         1630:	 //正极叠片升降移动至a等待高度 		  
	           			IF NOT DP_SinStepe THEN					
								 IF arrAxisCtrl[AxiseNo.AxisName.AnDTCarryingUpDown].Status.Homed AND arrAxisCtrl[AxiseNo.AxisName.AnDTCarryingUpDown].Status.NoMoving AND 
									NOT arrAxisCtrl[AxiseNo.AxisName.AnDTCarryingUpDown].Status.Error AND arrAxisCtrl[AxiseNo.AxisName.AnDTCarryingLine].Cmd.arrbRealPoint[2] AND
										 arrAxisCtrl[AxiseNo.AxisName.LeftYDUpDown].Cmd.arrbRealPoint[1] AND arrAxisCtrl[AxiseNo.AxisName.RightYDLine].Cmd.arrbRealPoint[2]     THEN
										IF arrAxisCtrl[AxiseNo.AxisName.AnDTCarryingUpDown].Cmd.arrbRealPoint[4] THEN
											arrAxisCtrl[AxiseNo.AxisName.AnDTCarryingUpDown].Cmd.iGoSetPos:=0;
										ELSE
											arrAxisCtrl[AxiseNo.AxisName.AnDTCarryingUpDown].Cmd.iGoSetPos:=4;//正极叠片升降移动至等待高度
										END_IF
								END_IF 
                                (*
								IF 	arrAxisCtrl[AxiseNo.AxisName.RightYDUpDown].Status.Homed AND arrAxisCtrl[AxiseNo.AxisName.RightYDUpDown].Status.NoMoving THEN
									IF arrAxisCtrl[AxiseNo.AxisName.RightYDUpDown].Cmd.arrbRealPoint[1] THEN
										arrAxisCtrl[AxiseNo.AxisName.RightYDUpDown].Cmd.iGoSetPos:=0;
									ELSE
										arrAxisCtrl[AxiseNo.AxisName.RightYDUpDown].Cmd.iGoSetPos:=1;//右压刀升降上升至初始高度
									END_IF
								END_IF													
  	                            *)
								IF arrAxisCtrl[AxiseNo.AxisName.AnDTCarryingUpDown].Cmd.arrbRealPoint[4] AND arrAxisCtrl[AxiseNo.AxisName.RightYDUpDown].Cmd.arrbRealPoint[15] AND
                                    arrAxisCtrl[AxiseNo.AxisName.AnDTCarryingUpDown].Status.NoMoving  AND arrAxisCtrl[AxiseNo.AxisName.RightYDUpDown].Status.NoMoving    THEN
						         	DT_SingeMode();//单步选择
									An_OverNGStep:=1670;
								END_IF		
                       END_IF	   						
 (*
  		1640://	压刀升降上升至初始高度	
					IF NOT DP_SinStepe THEN								
								IF 	arrAxisCtrl[AxiseNo.AxisName.RightYDUpDown].Status.Homed AND arrAxisCtrl[AxiseNo.AxisName.RightYDUpDown].Status.NoMoving THEN
									IF arrAxisCtrl[AxiseNo.AxisName.RightYDUpDown].Cmd.arrbRealPoint[1] THEN
										arrAxisCtrl[AxiseNo.AxisName.RightYDUpDown].Cmd.iGoSetPos:=0;
									ELSE
										arrAxisCtrl[AxiseNo.AxisName.RightYDUpDown].Cmd.iGoSetPos:=1;//右压刀升降上升至初始高度
									END_IF
								END_IF				
								IF arrAxisCtrl[AxiseNo.AxisName.RightYDUpDown].Cmd.arrbRealPoint[1] THEN
							     	DT_SingeMode();//单步选择
									An_OverNGStep:=1641;
								END_IF
						END_IF	   
	
		1641://	右压刀开合移至初始位		
			       IF NOT DP_SinStepe THEN
								IF 	arrAxisCtrl[AxiseNo.AxisName.RightYDLine].Status.Homed AND arrAxisCtrl[AxiseNo.AxisName.RightYDLine].Status.NoMoving THEN
										IF arrAxisCtrl[AxiseNo.AxisName.RightYDLine].Cmd.arrbRealPoint[1] THEN
											arrAxisCtrl[AxiseNo.AxisName.RightYDLine].Cmd.iGoSetPos:=0;
											DT_SingeMode();//单步选择
											An_OverNGStep:=1650;
										ELSE
											arrAxisCtrl[AxiseNo.AxisName.RightYDLine].Cmd.iGoSetPos:=1;//右压刀开合至初始位
										END_IF		
                                END_IF;	
					END_IF;				
					
		   	1650://右压刀升降下降至初始位，压隔膜			
					  IF NOT DP_SinStepe THEN
	                         	IF 	arrAxisCtrl[AxiseNo.AxisName.RightYDUpDown].Status.Homed AND arrAxisCtrl[AxiseNo.AxisName.RightYDUpDown].Status.NoMoving THEN
										IF arrAxisCtrl[AxiseNo.AxisName.RightYDUpDown].Cmd.arrbRealPoint[1] THEN
											arrAxisCtrl[AxiseNo.AxisName.RightYDUpDown].Cmd.iGoSetPos:=0;
									     	DT_SingeMode();//单步选择
									    	An_OverNGStep:=1670;
										ELSE
											arrAxisCtrl[AxiseNo.AxisName.RightYDUpDown].Cmd.iGoSetPos:=1;//右压刀升降轴下降至初始高度
										END_IF
									END_IF							  
					  
					  END_IF					   
					   
		     //1660:	 //判断真空					   
	*)

           1670://判断主轴是否停止、是否在初始位、是否有轴在耦合中
					IF NOT DP_SinStepe THEN
								IF arrAxis[AxiseNo.VirAxisName.VirMain].Status.NotMoving AND arrAxis[AxiseNo.VirAxisName.VirMain].NcToPlc.SetPos=0 AND NOT DT_AxiseCoupling THEN
									DT_SingeMode();//单步选择
									An_OverNGStep:=1691;
								ELSE
									DP_Step1:=100;//调用主轴回初始位子程序
									DT_SingeMode();//单步选择
									An_OverNGStep:=1690;
								END_IF
			    	END_IF		
			1690://判断主轴的模长的当前位置是否为0
				IF NOT DP_SinStepe THEN
					IF DP_Step1=6666 AND arrAxis[AxiseNo.VirAxisName.VirMain].Status.NotMoving AND arrAxis[AxiseNo.VirAxisName.VirMain].NcToPlc.SetPos=0 AND NOT DT_AxiseCoupling  THEN
						DT_SingeMode();//单步选择
						An_OverNGStep:=1691;
					END_IF	
				END_IF				
		1691:
			    IF 	arrAxisCtrl[AxiseNo.AxisName.LeftYDUpDown].Cmd.arrbRealPoint[1] AND (arrAxisCtrl[AxiseNo.AxisName.RightYDUpDown].Cmd.arrbRealPoint[1] OR arrAxisCtrl[AxiseNo.AxisName.RightYDUpDown].Cmd.arrbRealPoint[15] ) AND
					    arrCyCtrl[arrCyNo.CylinderName.AnScrapbinCy].Status.ONState  AND arrCyCtrl[arrCyNo.CylinderName.CaScrapbinUDCy].Status.OFFState AND
                        arrCyCtrl[arrCyNo.CylinderName.PoleHotCutterCy].Status.OFFState   THEN
					An_OverNGStep:=1695;
				END_IF	
		
		    1695://				
					IF An_CarryingPos2 THEN//正极在叠片位
							An_OverNGStep:=1700;//
					ELSIF An_CarryingPos1  THEN//正极在取片位
							 An_OverNGStep:=1800;//
					ELSE
						  DTPosError[11]:=TRUE;//踢正极对齐度NG片 时，正极取片即不在取片位，也不在叠片位
					END_IF;
		
	

	        1800://	调用正极NG踢废		
                    DT_TON[2].IN:=FALSE;	
					CCD.Over.Start.iPhotoDo:=2;
					CCD.Over.Finish.OverhandResult:=0;
					Mach_Control.DT_b.OverhandResult:=0;
					Mach_Control.DT_b.CDD_OverStart:=TRUE;
					
			        Mach_Control.An_b.An_Quantited:=Mach_Control.An_b.An_Quantited-1;//正极已叠片数减一
                    An_Step2:=10; 
                    An_OverNGStep:=1810;

			1810://判断负极叠台搬运是否有片，有片的话放到纠偏台
			         DT_TON[2].IN:=TRUE;	
						IF arrCyCtrl[arrCyNo.ElectValveName.CaDTCarryingVacuum].Io.DIOnSwitch AND  Mach_Control.Ca_b.Ca_DPCarryingFalg  THEN//负极再取片位且叠台搬运有片,把当前片放到纠偏台
							An_OverNGStep:=1820;
						ELSE
							An_OverNGStep:=1850;	
						END_IF
	
			1820://纠偏台回初始位
				//纠偏平台X1移动至初始位
				IF NOT DP_SinStepe THEN
					IF arrAxisCtrl[AxiseNo.AxisName.CadeviationX1].Status.Homed  AND arrAxisCtrl[AxiseNo.AxisName.CadeviationX1].Status.NoMoving AND NOT  arrAxisCtrl[AxiseNo.AxisName.CadeviationX1].Status.Error THEN
						IF arrAxisCtrl[AxiseNo.AxisName.CadeviationX1].Cmd.arrbRealPoint[1] THEN
							arrAxisCtrl[AxiseNo.AxisName.CadeviationX1].Cmd.iGoSetPos:=0;
						ELSE
							arrAxisCtrl[AxiseNo.AxisName.CadeviationX1].Cmd.iGoSetPos:=1;
						END_IF					
					END_IF
					//纠偏平台X2移动至初始位
					IF arrAxisCtrl[AxiseNo.AxisName.CadeviationX2].Status.Homed  AND arrAxisCtrl[AxiseNo.AxisName.CadeviationX2].Status.NoMoving AND NOT  arrAxisCtrl[AxiseNo.AxisName.CadeviationX2].Status.Error THEN
						IF arrAxisCtrl[AxiseNo.AxisName.CadeviationX2].Cmd.arrbRealPoint[1] THEN
							arrAxisCtrl[AxiseNo.AxisName.CadeviationX2].Cmd.iGoSetPos:=0;
						ELSE
							arrAxisCtrl[AxiseNo.AxisName.CadeviationX2].Cmd.iGoSetPos:=1;
						END_IF					
					END_IF
					//纠偏平台X2移动至初始位
					IF arrAxisCtrl[AxiseNo.AxisName.CadeviationY].Status.Homed  AND arrAxisCtrl[AxiseNo.AxisName.CadeviationY].Status.NoMoving AND NOT  arrAxisCtrl[AxiseNo.AxisName.CadeviationY].Status.Error THEN
						IF arrAxisCtrl[AxiseNo.AxisName.CadeviationY].Cmd.arrbRealPoint[1] THEN
							arrAxisCtrl[AxiseNo.AxisName.CadeviationY].Cmd.iGoSetPos:=0;
						ELSE
							arrAxisCtrl[AxiseNo.AxisName.CadeviationY].Cmd.iGoSetPos:=1;
						END_IF					
					END_IF
					IF arrAxisCtrl[AxiseNo.AxisName.CadeviationX1].Cmd.arrbRealPoint[1] AND arrAxisCtrl[AxiseNo.AxisName.CadeviationX2].Cmd.arrbRealPoint[1] AND arrAxisCtrl[AxiseNo.AxisName.CadeviationY].Cmd.arrbRealPoint[1] THEN
						DT_SingeMode();//单步选择	
						An_OverNGStep:=1830;	
						DT_TON[4].IN:=FALSE;
					END_IF	
				END_IF
			1830://叠台搬运极片放回纠偏台
				IF NOT DP_SinStepe THEN
					IF arrAxisCtrl[AxiseNo.AxisName.CaDTCarryingLine].Cmd.arrbRealPoint[1]  AND NOT Mach_Control.Ca_b.Ca_deviationFalg THEN 
						IF arrAxisCtrl[AxiseNo.AxisName.CaDTCarryingUpDown].Cmd.arrbRealPoint[2] THEN
							arrAxisCtrl[AxiseNo.AxisName.CaDTCarryingUpDown].Cmd.iGoSetPos:=0;
					    ELSE
							arrAxisCtrl[AxiseNo.AxisName.CaDTCarryingUpDown].Cmd.iGoSetPos:=2;//负极d叠台搬运下降至取片位
					    END_IF
                   END_IF
				       IF arrAxisCtrl[AxiseNo.AxisName.CaDTCarryingUpDown].Cmd.arrbRealPoint[2] THEN
				           	/// 吸盘破真空    纠偏台开真空
							arrCyCtrl[arrCyNo.ElectValveName.CaDTCarryingVacuum].Cmd.bON:=TRUE;	//负极叠台搬运升降真空	真空
							arrCyCtrl[arrCyNo.ElectValveName.CaDTCarryingVacuum].Cmd.bOFF:=FALSE;	//负极叠台搬运升降真空破真空								
							arrCyCtrl[arrCyNo.ElectValveName.CadeviationVacuum].Cmd.bON:=TRUE;	//负极纠偏台真空			
							arrCyCtrl[arrCyNo.ElectValveName.CadeviationVacuum].Cmd.bOFF:=FALSE;	//负极纠偏台真空	   
							DT_SingeMode();//单步选择	
							An_OverNGStep:=1840;
							DT_TON[4].IN:=TRUE;
							Mach_Control.Ca_b.Ca_deviationFalg:=TRUE;//置位位纠偏平台有料标记
							Mach_Control.Ca_b.Ca_DPCarryingFalg:=FALSE;//负极搬运真空吸盘有料标记复位
	                    END_IF
				END_IF
			1840://叠台搬运极片上升至凸轮耦合初始高度
				IF NOT DP_SinStepe THEN
					IF arrAxisCtrl[AxiseNo.AxisName.CaDTCarryingUpDown].Cmd.arrbRealPoint[4] AND DT_TON[4].Q THEN
						arrAxisCtrl[AxiseNo.AxisName.CaDTCarryingUpDown].Cmd.iGoSetPos:=0;
						/// 吸盘破真空    纠偏台开真空
						Mach_Control.Ca_b.Ca_deviationFalg:=TRUE;//置位位纠偏平台有料标记
						Mach_Control.Ca_b.Ca_DPCarryingFalg:=FALSE;//负极搬运真空吸盘有料标记复位
						Par.stDT_date.Ca_MQ_Slice[8]:=Par.stDT_date.Ca_MQ_Slice[9];
						DT_SingeMode();//单步选择	
						An_OverNGStep:=1850;
						DT_TON[4].IN:=FALSE;
					ELSE
						arrAxisCtrl[AxiseNo.AxisName.CaDTCarryingUpDown].Cmd.iGoSetPos:=4;//负极搬运升降2上升至凸轮耦合初始高度
					END_IF			
				END_IF		   
		

			
	        1860://等待正极NG踢废完成		
  
				
					 IF 	An_Step2=6666 THEN
						    An_OverNGStep:=0;
							DP_Step0:=0;
                           // An_OverNGMark:=FALSE;	
					 END_IF
	  END_CASE
END_IF

 CASE An_OverNGStep OF  
	 
		1850://
                  
				   IF Mach_Control.DT_b.OverhandResult<>3 AND  DT_TON[2].Q THEN
					  Mach_Control.An_b.Error[22]:=TRUE;//正极叠台搬运升降真空报警，电芯上有片，请拿掉 
				   END_IF
			
				 IF 	 Mach_Control.DT_b.OverhandResult=3 THEN
					     DT_TON[2].IN:=FALSE;	
						An_OverNGStep:=1860;
				 END_IF
 
 
 
 
     1200: //正到负取正极NG对其度片,	正极搬运与叠片各轴在初始位,负极在叠片位
	             VirMain_TON.IN:=FALSE;   
				//正到负_正极送片搬运平移轴凸轮耦合
				fbAnCamInCarryingLine.ParCamIn.SlaveScaling:=1;
				fbAnCamInCarryingLine.bCamInExecute:=TRUE;	
		    	fbAnCamInCarryingUpDown.iTableSel:=3;      //20240528SJ
                fbAnCamInCarryingUpDown.bCamInExecute:=TRUE;
			//正到负_正极叠片平移轴凸轮耦合
				fbAnCamInDTCarryingLine.ParCamIn.SlaveScaling:=1;
				fbAnCamInDTCarryingLine.bCamInExecute:=TRUE;			
                fbAnCamInDTCarryingUpDown.iTableSel:=3;   //  //20240528SJ
                fbAnCamInDTCarryingUpDown.bCamInExecute:=TRUE;
			//正到负_正极搬运旋转轴凸轮耦合		
				fbAnCamInCarryingWhirling.ParCamIn.SlaveScaling:=1;
				fbAnCamInCarryingWhirling.bCamInExecute:=TRUE;						
			
			//正到负_负极送片搬运平移轴凸轮耦合
				fbCaCamInCarryingLine2.ParCamIn.SlaveScaling:=-1;
				fbCaCamInCarryingLine2.bCamInExecute:=TRUE;
			   fbCaCamInCarryingUpDown2.iTableSel:=3; //20240528SJ
               fbCaCamInCarryingUpDown2.bCamInExecute:=TRUE;
			//正到负_负极叠片搬运平移轴凸轮耦合
				fbCaCamInDTCarryingLine.ParCamIn.SlaveScaling:=-1;
				fbCaCamInDTCarryingLine.bCamInExecute:=TRUE;
			    fbCaCamInDTCarryingUpDown.iTableSel:=3;  //20240528SJ
                fbCaCamInDTCarryingUpDown.bCamInExecute:=TRUE;
			//正到负_ 缓存轴轮耦合
				fbCamInGMBuffer2.iTableSel:=1;
				 fbCamInGMBuffer2.bCamInExecute:=TRUE;
			//正到负_隔膜平移轴凸轮耦合
				fbCamInGMDanserMove.iTableSel:=1;
				fbCamInGMDanserMove.bCamInExecute:=TRUE;
			
			//正到负_放卷虚轴凸轮耦合
				 fbCamInVirGMDriver2.iTableSel :=1;
				 fbCamInVirGMDriver2.bCamInExecute:=TRUE;		
					
					//判断凸轮是否耦合完成
						IF  fbAnCamInCarryingLine.bInSync  AND  fbAnCamInDTCarryingLine.bInSync AND fbAnCamInCarryingWhirling.bInSync AND 
							 fbCaCamInCarryingLine2.bInSync AND fbCaCamInDTCarryingLine.bInSync AND
							 fbCamInGMBuffer2.bInSync AND fbCamInGMDanserMove.bInSync AND 
							 fbCamInVirGMDriver2.bInSync   AND
							 fbAnCamInCarryingUpDown.bInSync AND fbAnCamInDTCarryingUpDown.bInSync AND fbCaCamInCarryingUpDown2.bInSync AND fbCaCamInDTCarryingUpDown.bInSync AND  
                            Mach_Control.U.DT_iMode=1  THEN
							An_OverNGStep:=1210;//
						ELSIF   fbAnCamInCarryingLine.bError  OR  fbAnCamInDTCarryingLine.bError OR 
							 fbCaCamInCarryingLine2.bError OR fbCaCamInDTCarryingLine.bError OR
							 fbCamInGMBuffer2.bError OR fbCamInGMDanserMove.bError OR 
							  fbAnCamInCarryingUpDown.bError OR fbAnCamInDTCarryingUpDown.bError OR fbCaCamInCarryingUpDown2.bError OR fbCaCamInDTCarryingUpDown.bError OR  
							 fbCamInVirGMDriver2.bError THEN
								Mach_Control.DT_b.Error[19]:=TRUE;//凸轮耦合报警
								An_OverNGStep:=9991;										
						END_IF		
			1210://主轴启动
									arrAxisCtrl[AxiseNo.VirAxisName.VirMain].Cmd	.bDynamitcsParSel:=2;
									arrAxisPar[AxiseNo.VirAxisName.VirMain].fTagatTime:=VirMain_TagatTime;
									arrAxisCtrl[AxiseNo.VirAxisName.VirMain].Cmd	.fPositon_of_Abs:=360;
									arrAxisCtrl[AxiseNo.VirAxisName.VirMain].Cmd	.bMoveAbs:=TRUE;		
									
									IF  arrAxis[AxiseNo.VirAxisName.VirMain].Status.Moving AND arrAxisCtrl[AxiseNo.VirAxisName.VirMain].Status.fActPos>=10  THEN
										VirMain_TON.IN:=FALSE;
										arrAxisCtrl[AxiseNo.VirAxisName.VirMain].Cmd	.bMoveAbs:=FALSE;	
										An_OverNGStep:=1500;	
									ELSE
										IF NOT VirMain_TON.Q THEN
											VirMain_TON.IN:=TRUE;
										ELSE
											VirMain_TON.IN:=FALSE;
											Mach_Control.DT_b.Error[22]:=TRUE;//主轴启动超时报警
											An_OverNGStep:=10001;	
									END_IF	
				 	    END_IF		

           1300: //正到负取正极NG对其度片,正极搬运与叠片各轴在初始位,, 负极在取片位,  隔膜平移在负极位
		              VirMain_TON.IN:=FALSE;
						//正到负_正极送片搬运平移轴凸轮耦合
					fbAnCamInCarryingLine.ParCamIn.SlaveScaling:=1;
					fbAnCamInCarryingLine.bCamInExecute:=TRUE;					
					fbAnCamInCarryingUpDown.iTableSel:=3;      //20240528SJ
					fbAnCamInCarryingUpDown.bCamInExecute:=TRUE;
				//正到负_正极叠片平移轴凸轮耦合
					fbAnCamInDTCarryingLine.ParCamIn.SlaveScaling:=1;
					fbAnCamInDTCarryingLine.bCamInExecute:=TRUE;		
					fbAnCamInDTCarryingUpDown.iTableSel:=3;   //  //20240528SJ
					fbAnCamInDTCarryingUpDown.bCamInExecute:=TRUE;

			//正到负_正极搬运旋转轴凸轮耦合		
				fbAnCamInCarryingWhirling.ParCamIn.SlaveScaling:=1;
				fbAnCamInCarryingWhirling.bCamInExecute:=TRUE;							
								
					//判断凸轮是否耦合完成
						IF  fbAnCamInCarryingLine.bInSync AND fbAnCamInDTCarryingLine.bInSync AND  fbAnCamInCarryingWhirling.bInSync  AND 
                            fbAnCamInCarryingUpDown.bInSync AND  fbAnCamInDTCarryingUpDown.bInSync AND 
                            Mach_Control.U.DT_iMode=1 THEN
							An_OverNGStep:=1310;//
						ELSIF fbAnCamInCarryingLine.bError OR  fbAnCamInDTCarryingLine.bError  OR   fbAnCamInCarryingUpDown.bError OR   fbAnCamInDTCarryingUpDown.bError   THEN
								Mach_Control.DT_b.Error[19]:=TRUE;//凸轮耦合报警
								An_OverNGStep:=9992;										
						END_IF			   
		   
			1310://主轴启动
									arrAxisCtrl[AxiseNo.VirAxisName.VirMain].Cmd	.bDynamitcsParSel:=2;
									arrAxisPar[AxiseNo.VirAxisName.VirMain].fTagatTime:=VirMain_TagatTime;
									arrAxisCtrl[AxiseNo.VirAxisName.VirMain].Cmd	.fPositon_of_Abs:=360;
									arrAxisCtrl[AxiseNo.VirAxisName.VirMain].Cmd	.bMoveAbs:=TRUE;			
						
									IF  arrAxis[AxiseNo.VirAxisName.VirMain].Status.Moving AND arrAxisCtrl[AxiseNo.VirAxisName.VirMain].Status.fActPos>=10  THEN
										VirMain_TON.IN:=FALSE;
										arrAxisCtrl[AxiseNo.VirAxisName.VirMain].Cmd	.bMoveAbs:=FALSE;	
										An_OverNGStep:=1500;	
									ELSE
										IF NOT VirMain_TON.Q THEN
											VirMain_TON.IN:=TRUE;
										ELSE
											VirMain_TON.IN:=FALSE;
											Mach_Control.DT_b.Error[22]:=TRUE;//主轴启动超时报警
											An_OverNGStep:=10002;	
									END_IF	
				 	    END_IF							
										
	       1400: //正到负取正极NG对其度片,正极搬运与叠片各轴在初始位,, 负极在取片位,  隔膜平移在正极位	
			              VirMain_TON.IN:=FALSE;
						//正到负_正极送片搬运平移轴凸轮耦合
						fbAnCamInCarryingLine.ParCamIn.SlaveScaling:=1;
						fbAnCamInCarryingLine.bCamInExecute:=TRUE;				
						fbAnCamInCarryingUpDown.iTableSel:=3;      //20240528SJ
						fbAnCamInCarryingUpDown.bCamInExecute:=TRUE;

					//正到负_正极叠片平移轴凸轮耦合
						fbAnCamInDTCarryingLine.ParCamIn.SlaveScaling:=1;
						fbAnCamInDTCarryingLine.bCamInExecute:=TRUE;
					   fbAnCamInDTCarryingUpDown.iTableSel:=3;   //  //20240528SJ
                       fbAnCamInDTCarryingUpDown.bCamInExecute:=TRUE;
						
						
					//正到负_正极搬运旋转轴凸轮耦合		
						fbAnCamInCarryingWhirling.ParCamIn.SlaveScaling:=1;
						fbAnCamInCarryingWhirling.bCamInExecute:=TRUE;						
						
					//正到负_ 缓存轴轮耦合
						fbCamInGMBuffer2.iTableSel:=1;
						 fbCamInGMBuffer2.bCamInExecute:=TRUE;
						 
					//正到负_隔膜平移轴凸轮耦合
						fbCamInGMDanserMove.iTableSel:=1;
						fbCamInGMDanserMove.bCamInExecute:=TRUE;
						
					//正到负_放卷虚轴凸轮耦合
						 fbCamInVirGMDriver2.iTableSel :=1;
						 fbCamInVirGMDriver2.bCamInExecute:=TRUE;			   
						
					//判断凸轮是否耦合完成
						IF   fbAnCamInCarryingLine.bInSync  AND  fbAnCamInDTCarryingLine.bInSync AND   fbAnCamInCarryingWhirling.bInSync AND
							 fbCamInGMBuffer2.bInSync AND fbCamInGMDanserMove.bInSync AND 
							 fbAnCamInCarryingUpDown.bInSync AND fbAnCamInDTCarryingUpDown.bInSync AND 
							 fbCamInVirGMDriver2.bInSync  AND 
                            Mach_Control.U.DT_iMode=1  THEN
							An_OverNGStep:=1410;//
						ELSIF  fbAnCamInCarryingLine.bError  OR  fbAnCamInDTCarryingLine.bError OR 
							     fbCamInGMBuffer2.bError OR fbCamInGMDanserMove.bError OR 
								 fbAnCamInCarryingUpDown.bError OR  fbAnCamInDTCarryingUpDown.bError OR
							     fbCamInVirGMDriver2.bError THEN
										Mach_Control.DT_b.Error[19]:=TRUE;//凸轮耦合报警
										An_OverNGStep:=9993;										
						END_IF		
	
			1410://主轴启动
									arrAxisCtrl[AxiseNo.VirAxisName.VirMain].Cmd	.bDynamitcsParSel:=2;
									arrAxisPar[AxiseNo.VirAxisName.VirMain].fTagatTime:=VirMain_TagatTime;
									arrAxisCtrl[AxiseNo.VirAxisName.VirMain].Cmd	.fPositon_of_Abs:=360;
									arrAxisCtrl[AxiseNo.VirAxisName.VirMain].Cmd	.bMoveAbs:=TRUE;					
									IF  arrAxis[AxiseNo.VirAxisName.VirMain].Status.Moving AND arrAxisCtrl[AxiseNo.VirAxisName.VirMain].Status.fActPos>=10  THEN
										VirMain_TON.IN:=FALSE;
										arrAxisCtrl[AxiseNo.VirAxisName.VirMain].Cmd	.bMoveAbs:=FALSE;	
										An_OverNGStep:=1500;	
									ELSE
										IF NOT VirMain_TON.Q THEN
											VirMain_TON.IN:=TRUE;
										ELSE
											VirMain_TON.IN:=FALSE;
											Mach_Control.DT_b.Error[22]:=TRUE;//主轴启动超时报警
											An_OverNGStep:=10003;	
									END_IF	
				 	    END_IF							
   
			1500://
				(*IF 	arrAxisCtrl[AxiseNo.VirAxisName.VirMain].Status.fActPos>230 AND  arrAxisCtrl[AxiseNo.VirAxisName.VirMain].Status.fActPos<240 AND Mach_Control.Ca_b.Ca_DPCarryingFalg  THEN//198
					IF Mach_Control.DT_b.DT_CCD_TwoModel THEN
							CCD.CaRec.Finish.RectifyX1:=0;
							CCD.CaRec.Finish.RectifyX2:=0;
							CCD.CaRec.Finish.RectifyY:=0;		
							CCD.CaRec.Finish.RectifyResult:=0;//拍照结果清零									
							Mach_Control.Ca_b.Ca_CCDStart :=TRUE;//启动CCD拍照
							CCD.CaRec.Start.iPhotoDo:=2;//启动CCD第二次拍照									
					END_IF			
				END_IF	*)		
				
				IF arrAxis[AxiseNo.VirAxisName.VirMain].NcToPlc.SetPos=360 AND  arrAxis[AxiseNo.VirAxisName.VirMain].Status.NotMoving  THEN
					DP_Step1:=100;//解除耦合，主轴回零子程序			
					An_OverNGStep:=1510;	
				END_IF	
			1510://			
				IF NOT DP_SinStepe THEN
					IF DP_Step1=6666 AND arrAxis[AxiseNo.VirAxisName.VirMain].Status.NotMoving AND arrAxis[AxiseNo.VirAxisName.VirMain].NcToPlc.SetPos=0 AND NOT DT_AxiseCoupling  THEN
						DT_SingeMode();//单步选择
						An_OverNGStep:=1600;
					END_IF	
				END_IF	

		    1700://	/踢正极NG对齐度片回正极取片位,(正极轴不动 ) ,正极搬运叠片各轴在叠片位		
			         VirMain_TON.IN:=FALSE;
					//负到正_正极搬运平移轴凸轮耦合
					fbAnCamInCarryingLine.ParCamIn.SlaveScaling:=-1;
					fbAnCamInCarryingLine.bCamInExecute:=TRUE;
					fbAnCamInCarryingUpDown.iTableSel:=3;      //20240528SJ
                   fbAnCamInCarryingUpDown.bCamInExecute:=TRUE;
					
					//负到正_正极叠片平移轴凸轮耦合
					fbAnCamInDTCarryingLine.ParCamIn.SlaveScaling:=-1;
					fbAnCamInDTCarryingLine.bCamInExecute:=TRUE;	
					fbAnCamInDTCarryingUpDown.iTableSel:=3;   //  //20240528SJ
					fbAnCamInDTCarryingUpDown.bCamInExecute:=TRUE;

					//负到正_正极搬运旋转轴凸轮耦合
						fbAnCamInCarryingWhirling.ParCamIn.SlaveScaling:=-1;
						fbAnCamInCarryingWhirling.bCamInExecute:=TRUE;								
				
				IF fbAnCamInCarryingLine.bInSync  AND 
					fbAnCamInDTCarryingLine.bInSync  AND
					fbAnCamInCarryingWhirling.bInSync AND  
                    fbAnCamInCarryingUpDown.bInSync AND   fbAnCamInDTCarryingUpDown.bInSync AND  
                    Mach_Control.U.DT_iMode=1  THEN   
					DT_SingeMode();//单步选择		
					An_OverNGStep:=1710;
				ELSIF fbAnCamInCarryingLine.bError OR //  fbCaCamInCarryingUpDown2.bError or
					  fbAnCamInDTCarryingLine.bError  OR  fbAnCamInCarryingUpDown.bError OR    fbAnCamInDTCarryingUpDown.bError   THEN   
					Mach_Control.DT_b.Error[19]:=TRUE;//凸轮耦合报警
					An_OverNGStep:=9994;
				END_IF		

				1710://主轴启动
				      				
									arrAxisCtrl[AxiseNo.VirAxisName.VirMain].Cmd	.bDynamitcsParSel:=2;
									arrAxisPar[AxiseNo.VirAxisName.VirMain].fTagatTime:=VirMain_TagatTime;
									arrAxisCtrl[AxiseNo.VirAxisName.VirMain].Cmd	.fPositon_of_Abs:=360;
									arrAxisCtrl[AxiseNo.VirAxisName.VirMain].Cmd	.bMoveAbs:=TRUE;			
						IF  arrAxis[AxiseNo.VirAxisName.VirMain].Status.Moving AND arrAxisCtrl[AxiseNo.VirAxisName.VirMain].Status.fActPos>=10  THEN
							VirMain_TON.IN:=FALSE;
							arrAxisCtrl[AxiseNo.VirAxisName.VirMain].Cmd	.bMoveAbs:=FALSE;	
							An_OverNGStep:=1720;	
						ELSE
								IF NOT VirMain_TON.Q THEN
									VirMain_TON.IN:=TRUE;
								ELSE
									VirMain_TON.IN:=FALSE;
									Mach_Control.DT_b.Error[22]:=TRUE;//主轴启动超时报警
									An_OverNGStep:=10004;	
							END_IF	
					   END_IF				

			1720://
				IF arrAxis[AxiseNo.VirAxisName.VirMain].NcToPlc.SetPos=360 AND  arrAxis[AxiseNo.VirAxisName.VirMain].Status.NotMoving  THEN
					DP_Step1:=100;//解除耦合，主轴回零子程序			
					An_OverNGStep:=1730;	
				END_IF	
	
				
			1730://			
				IF NOT DP_SinStepe THEN
					IF DP_Step1=6666 AND arrAxis[AxiseNo.VirAxisName.VirMain].Status.NotMoving AND arrAxis[AxiseNo.VirAxisName.VirMain].NcToPlc.SetPos=0 AND NOT DT_AxiseCoupling  THEN
						DT_SingeMode();//单步选择
						An_OverNGStep:=1800;
					END_IF	
				END_IF	
									
 END_CASE
END_ACTION

ACTION An_Rectifydev:
rAnCCD_Ton(IN:= , PT:=T#1.5S , Q=> , ET=> );//正极CCD拍照超时报警
IF (NOT Mach_Control.An_b.An_deviationFalg AND Mach_Control.U.DT_iMode=1) AND NOT Mach_Control.An_b.Demarcateing   THEN
//IF NOT Mach_Control.An_b.An_deviationFalg THEN
	Mach_Control.An_b.RectifydevDone:=FALSE;
	An_CCD_Done:=FALSE;
	CCD.AnRec.Finish.RectifyX1:=0;
	CCD.AnRec.Finish.RectifyX2:=0;
	CCD.AnRec.Finish.RectifyY:=0;
END_IF

rAnCCD_Ton1(IN:=Mach_Control.An_b.An_CCDStart , PT:=T#0.1S , Q=> , ET=> );//正极CCD拍照启动复位
IF rAnCCD_Ton1.Q THEN
	Mach_Control.An_b.An_CCDStart :=FALSE;
END_IF


An_CQ_ton(IN:=arrCyCtrl[arrCyNo.ElectValveName.AndeviationIonizedWind].Io.DOStatus1 , PT:=T#0.3S , Q=> , ET=>);
IF An_CQ_ton.Q THEN
	Mach_Control.An_b.An_Rectifydev_CQ:=FALSE;
	arrCyCtrl[arrCyNo.ElectValveName.AndeviationIonizedWind].Cmd.bON:=FALSE;//正极纠偏平台除尘
	arrCyCtrl[arrCyNo.ElectValveName.AndeviationIonizedWind].Cmd.bOFF:=TRUE;//正极纠偏平台除尘
END_IF



IF rAnUse[2].Q THEN
	CCD.AnRec.Finish.RectifyResult:=0;
	CCD.AnRec.Finish.RectifyX1:=0;
	CCD.AnRec.Finish.RectifyX2:=0;
	CCD.AnRec.Finish.RectifyY:=0;												
END_IF



IF Mach_Control.U.DT_iMode=1 THEN//在自动状态下
//判断负极是否允许取纠偏
IF (Mach_Control.An_b.An_deviationFalg AND (An_CCD_Done OR Mach_Control.An_b.RectifydevDone)) (*AND CCD.AnRec.Finish.RectifyResult=1 AND Mach_Control.An_b.RectifydevDone)*) OR
	 (Mach_Control.An_b.An_deviationFalg AND CCD.AnRec.Finish.RectifyResult<>1 AND arrAxisCtrl[AxiseNo.AxisName.AndeviationX1].Cmd.arrbRealPoint[1] AND 	arrAxisCtrl[AxiseNo.AxisName.AndeviationX2].Cmd.arrbRealPoint[1]  AND 	arrAxisCtrl[AxiseNo.AxisName.AndeviationY].Cmd.arrbRealPoint[1] )OR
	(Mach_Control.U.CCD_ChosesHMI  OR Mach_Control.U.EmptyRunMode)	 THEN
	Mach_Control.An_b.An_deviationDPOK:=TRUE;//取正极 偏平台极片允许
ELSE
	Mach_Control.An_b.An_deviationDPOK:=FALSE;
END_IF 	

	CASE An_StandbyStep0 OF
			0://判断正极纠偏平台是否有极片
				IF Mach_Control.An_b.An_deviationFalg AND NOT Mach_Control.U.EmptyRunMode  THEN
						IF NOT An_CCD_Done THEN
							CCD.AnRec.Finish.RectifyResult:=0;
							CCD.AnRec.Finish.RectifyX1:=0;
							CCD.AnRec.Finish.RectifyX2:=0;
							CCD.AnRec.Finish.RectifyY:=0;
							iMD11:=1;
							An_StandbyStep0:=10;
						END_IF
				ELSE
						iMD11:=2;
						An_RecdevPla_Step0:=0;
						Mach_Control.An_b.RectifydevStart :=FALSE;
						An_StandbyStep0:=10;
				END_IF
			10://正极纠偏平台回初始位
			IF  NOT Mach_Control.U.EmptyRunMode THEN
					Mach_Control.An_b.RectifydevStart :=FALSE;//复位纠偏启动
					Mach_Control.An_b.RectifydevDone:=FALSE;//复位纠偏完成
					IF Mach_Control.An_b.CarryingSafepos[4] THEN
							//纠偏平台X1移动至初始位
							IF arrAxisCtrl[AxiseNo.AxisName.AndeviationX1].Status.Homed  AND arrAxisCtrl[AxiseNo.AxisName.AndeviationX1].Status.NoMoving AND NOT  arrAxisCtrl[AxiseNo.AxisName.AndeviationX1].Status.Error THEN
								IF arrAxisCtrl[AxiseNo.AxisName.AndeviationX1].Cmd.arrbRealPoint[1] THEN
									arrAxisCtrl[AxiseNo.AxisName.AndeviationX1].Cmd.iGoSetPos:=0;
								ELSE
									arrAxisCtrl[AxiseNo.AxisName.AndeviationX1].Cmd.iGoSetPos:=1;
								END_IF					
							END_IF
							//纠偏平台X2移动至初始位
							IF arrAxisCtrl[AxiseNo.AxisName.AndeviationX2].Status.Homed  AND arrAxisCtrl[AxiseNo.AxisName.AndeviationX2].Status.NoMoving AND NOT  arrAxisCtrl[AxiseNo.AxisName.AndeviationX2].Status.Error THEN
								IF arrAxisCtrl[AxiseNo.AxisName.AndeviationX2].Cmd.arrbRealPoint[1] THEN
									arrAxisCtrl[AxiseNo.AxisName.AndeviationX2].Cmd.iGoSetPos:=0;
								ELSE
									arrAxisCtrl[AxiseNo.AxisName.AndeviationX2].Cmd.iGoSetPos:=1;
								END_IF					
							END_IF
							//纠偏平台X2移动至初始位
							IF arrAxisCtrl[AxiseNo.AxisName.AndeviationY].Status.Homed  AND arrAxisCtrl[AxiseNo.AxisName.AndeviationY].Status.NoMoving AND NOT  arrAxisCtrl[AxiseNo.AxisName.AndeviationY].Status.Error THEN
								IF arrAxisCtrl[AxiseNo.AxisName.AndeviationY].Cmd.arrbRealPoint[1] THEN
									arrAxisCtrl[AxiseNo.AxisName.AndeviationY].Cmd.iGoSetPos:=0;
								ELSE
									arrAxisCtrl[AxiseNo.AxisName.AndeviationY].Cmd.iGoSetPos:=1;
								END_IF					
							END_IF	
							IF 	 arrAxisCtrl[AxiseNo.AxisName.AndeviationX1].Cmd.arrbRealPoint[1] AND 	arrAxisCtrl[AxiseNo.AxisName.AndeviationX2].Cmd.arrbRealPoint[1]  AND 	arrAxisCtrl[AxiseNo.AxisName.AndeviationY].Cmd.arrbRealPoint[1] THEN
									IF  iMD11=1 THEN
											 An_StandbyStep0:=101;
											 rAnCCD_Ton.IN:=FALSE;
									 ELSIF  iMD11=2 THEN
											An_StandbyStep0:=0;
									 END_IF  			
							END_IF						
					END_IF
	END_IF
			101:
					CCD.AnRec.Finish.RectifyResult:=0;
					Mach_Control.An_b.An_CCDStart :=TRUE;//启动CCD拍照						
					CCD.AnRec.Start.iPhotoDo:=1;//第一次拍照	
					CCD.AnRec.Start.stPoleNo:=Par.stDT_date.An_MQ_Slice[1].stPoleNo;	
					An_StandbyStep0:=110;	
			110:
					IF NOT rAnCCD_Ton.Q THEN						
						rAnCCD_Ton.IN:=TRUE;
						IF Mach_Control.An_b.An_deviationCCDDone OR Mach_Control.U.CCD_ChosesHMI THEN
							rAnCCD_Ton.IN:=FALSE;
							An_CCD_Done:=TRUE;
							An_StandbyStep0:=111;
						END_IF
					ELSE
							rAnCCD_Ton.IN:=FALSE;
							Mach_Control.An_b.Error[7]:=TRUE;//正极CCD第一次拍照超时
							An_StandbyStep0:=9999;
					END_IF
			
			111://启动拍照			
					Mach_Control.An_b.An_CCDStart :=FALSE;//启动CCD拍照						
					rAnCCD_Ton.IN:=FALSE;
					An_StandbyStep0:=0;					

	END_CASE
ELSE
//正极纠偏平台CCD标定自动
IF Mach_Control.An_b.DemarcateStart THEN
	CCD.AnRec.Start.iPhotoDo:=1;//第一次拍照	
END_IF
An_Demarcate(
	Step0:=An_Demarcate_Step0,
	AxisX1_NO:=AxiseNo.AxisName.AndeviationX1 , //正极纠偏X1轴号
	AxisX2_NO:=AxiseNo.AxisName.AndeviationX2 , //正极纠偏X2轴号
	AxisY_NO:=AxiseNo.AxisName.AndeviationY , //正极纠偏Y轴号
	DemarcateStart:=Mach_Control.An_b.DemarcateStart , //纠偏平台CCD标定启动
	CCDStart:=Mach_Control.An_b.An_CCDStart , //CCD拍照启动
	CCDNo:=CCD.AnRec.iDemCount,//CCD拍照次数
	DemarcateResult:=CCD.AnRec.iDemarcatResult,//标定结果
	DemarcateDone:=Mach_Control.An_b.DemarcateDone ,//CCD标定完成
	Demarcateing:=Mach_Control.An_b.Demarcateing,	//CCD标定中
	Error :=Mach_Control.An_b.Error[8]  );//CCD标定NG
END_IF
//正极纠偏自动
rAn_RecdevPlaR_TRIG(CLK:=Mach_Control.An_b.An_deviationFalg AND (CCD.AnRec.Finish.RectifyResult=1 OR CCD.AnRec.Finish.RectifyResult=2 ) AND NOT Mach_Control.U.CCD_ChosesHMI AND NOT Mach_Control.An_b.RectifydevDone AND 
										 		(CCD.AnRec.Finish.RectifyX1<>0 OR CCD.AnRec.Finish.RectifyX2<>0 OR CCD.AnRec.Finish.RectifyY<>0) AND CCD.AnRec.Start.iPhotoDo=1  , Q=> );//AND NOT Mach_Control.An_b.An_VacuumErrorNG
IF rAn_RecdevPlaR_TRIG.Q  THEN//AND NOT Blueflaging
	Mach_Control.An_b.RectifydevStart:=TRUE;
END_IF

//纠偏结果限定
IF (CCD.AnRec.Finish.RectifyX1>=15 OR CCD.AnRec.Finish.RectifyX2>=15 OR CCD.AnRec.Finish.RectifyY>=10 OR
	CCD.AnRec.Finish.RectifyX1<=-15 OR CCD.AnRec.Finish.RectifyX2<=-15 OR CCD.AnRec.Finish.RectifyY<=-10) AND NOT Mach_Control.An_b.Demarcateing THEN
	CCD.AnRec.Finish.RectifyX1:=0;
	CCD.AnRec.Finish.RectifyX2:=0;
	CCD.AnRec.Finish.RectifyY:=0;
END_IF


CCD.AnRec.Finish.Offset_X:=fCaOffsetMean_X;
CCD.AnRec.Finish.Offset_Y:=fCaOffsetMean_Y;

An_RecdevPla(
	Step0:=An_RecdevPla_Step0,
	RecdevStart:=Mach_Control.An_b.RectifydevStart , //正极纠偏平台纠偏启动
	RecdevDone:=Mach_Control.An_b.RectifydevDone , //正极纠偏平台纠偏完成
	RecdevAgree:=Mach_Control.An_b.CarryingSafepos[4] , //正极纠偏平台纠偏允许
	AxisX1_NO:=AxiseNo.AxisName.AndeviationX1  , //正极纠偏平台X1轴号
	AxisX2_NO:=AxiseNo.AxisName.AndeviationX2 , //正极纠偏平台X2轴号
	AxisY_NO:=AxiseNo.AxisName.AndeviationY  , //正极纠偏平台Y轴号
	CCD_X1:=CCD.AnRec.Finish.RectifyX1 ,//正极纠偏平台X1纠偏量
	CCD_X2:=CCD.AnRec.Finish.RectifyX2 , //正极纠偏平台X2纠偏量
	CCD_Y:=CCD.AnRec.Finish.RectifyY );//正极纠偏平台Y纠偏量
	
//纠偏平台重复精度测试
AN_RectifyTry_fb(
	Execute:=Mach_Control.An_b.RectifyTryStart AND Mach_Control.U.DT_iMode=3 , //纠偏平台重复精度测试启动 
	AxisNO_X:=AxiseNo.AxisName.AndeviationX1 , 
	AxisNO_Y:= AxiseNo.AxisName.AndeviationX2, 
	AxisNO_R:=AxiseNo.AxisName.AndeviationY , 
	Demarcate_X:=Par.stDT_date.An_Demarcate_X , //纠偏平台重复精度测试X纠偏量
	Demarcate_Y:=Par.stDT_date.An_Demarcate_Y , //纠偏平台重复精度测试Y纠偏量
	Demarcate_R:=Par.stDT_date.An_Demarcate_R ,  //纠偏平台重复精度测试R纠偏量
	CCDNo:=Par.stDT_date.An_CCDNo, //纠偏平台重复精度测试次数
	CCDStart:= Mach_Control.An_b.An_CCDStart );
	
//吸盘重复精度测试		
An_SuckerTest_fb(
	Execute:=Mach_Control.An_b.SuckerTestStart AND Mach_Control.U.DT_iMode=3 , //吸盘重复精度测试启动 , 
	AxisNO_1:= AxiseNo.AxisName.AnDTCarryingUpDown, 
	AxisNO_2:=AxiseNo.AxisName.AnDTCarryingLine , 
	AxisNO_X:= AxiseNo.AxisName.AndeviationX1 , 
	AxisNO_Y:= AxiseNo.AxisName.AndeviationX2, 
	AxisNO_R:= AxiseNo.AxisName.AndeviationY , 
	DTCarryingVacuum:=arrCyNo.ElectValveName.AnDTCarryingVacuum , 
	deviationVacuum:= arrCyNo.ElectValveName.AndeviationVacuum, 
	deviationVacuumBark:=arrCyNo.ElectValveName.AndeviationVacuumBark, 
	CCDCount:= Par.stDT_date.An_CCDCount, //吸盘重复精度测试次数
	CCDStart:=Mach_Control.An_b.An_CCDStart,	
	CCD_X1:=CCD.AnRec.Finish.RectifyX1 ,//正极纠偏平台X1纠偏量
	CCD_X2:=CCD.AnRec.Finish.RectifyX2 , //正极纠偏平台X2纠偏量
	CCD_Y:=CCD.AnRec.Finish.RectifyY,//正极纠偏平台Y纠偏量
    DTiMode:= Mach_Control.U.DT_iMode  );
	
	//正极通讯监控
rtAn_CCDTest1(CLK:=Mach_Control.An_b.bAnCCD_TestDo , Q=> );
IF rtAn_CCDTest1.Q THEN
	bAn_CCDTest1:=FALSE;
	bAn_CCDTest2:=FALSE;
END_IF
IF Mach_Control.An_b.bAnCCD_TestDo THEN
	rtAn_CCDTest2(CLK:=Mach_Control.An_b.An_CCDStart , Q=> );
	rtAn_CCDTest3(CLK:=CCD.AnRec.Finish.RectifyResult<>0 , Q=> );
	rtAn_CCDTest4(CLK:=Mach_Control.An_b.An_deviationCCDDone , Q=> );
	IF rtAn_CCDTest2.Q THEN
		bAn_CCDTest1:=TRUE;
		bAn_CCDTest2:=TRUE;
		CCD.AnRec.Finish.RectifyResult:=0;
	END_IF
	IF rtAn_CCDTest3.Q THEN
		bAn_CCDTest1:=FALSE;
	END_IF	
	IF rtAn_CCDTest4.Q THEN
		bAn_CCDTest2:=FALSE;
	END_IF
	tonAn_CCDTest1(IN:=bAn_CCDTest1 , PT:=T#999MS , Q=> , ET=> );
	tonAn_CCDTest2(IN:=bAn_CCDTest2 , PT:=T#999MS , Q=> , ET=> );
	IF bAn_CCDTest1 THEN
		Mach_Control.An_b.iAnCCD_RectifyCT:= TIME_TO_INT(tonAn_CCDTest1.ET);
	END_IF
	IF bAn_CCDTest2 THEN
		Mach_Control.An_b.iAnCCD_PhotoCT:= TIME_TO_INT(tonAn_CCDTest2.ET);
	END_IF
	IF tonAn_CCDTest1.Q THEN
		Mach_Control.An_b.bAnCCD_TestDo:=FALSE;
	END_IF
END_IF
	
//正极白班NG计数
IF HMI_Hour>=8 AND HMI_Hour<20 AND An_Step2>50 AND An_Step2<70 THEN
  IF CCD.AnRec.Finish.NG_Code = 1 THEN
   CCD.AnRec.DayNgclassification.X1_NG :=CCD.AnRec.DayNgclassification.X1_NG+1 ;
   CCD.AnRec.Finish.NG_Code := 0 ;
  ELSIF CCD.AnRec.Finish.NG_Code = 2 THEN
   CCD.AnRec.DayNgclassification.X2_NG := CCD.AnRec.DayNgclassification.X2_NG+1 ;  
   CCD.AnRec.Finish.NG_Code := 0 ;
  ELSIF CCD.AnRec.Finish.NG_Code = 3 THEN
   CCD.AnRec.DayNgclassification.Y_NG := CCD.AnRec.DayNgclassification.Y_NG+1 ;  
   CCD.AnRec.Finish.NG_Code := 0 ;
  ELSIF CCD.AnRec.Finish.NG_Code = 4 THEN
   CCD.AnRec.DayNgclassification.R_NG := CCD.AnRec.DayNgclassification.R_NG+1 ;   
   CCD.AnRec.Finish.NG_Code := 0 ; 
  ELSIF CCD.AnRec.Finish.NG_Code = 5 THEN 
   CCD.AnRec.DayNgclassification.other_NG :=  CCD.AnRec.DayNgclassification.other_NG+1;
   CCD.AnRec.Finish.NG_Code := 0 ;
  END_IF	
END_IF  

DayClear1(CLK:=(HMI_Hour=8 AND HMI_Minute=0 AND HMI_Second=0 ) , Q=> );
NightClear1(CLK:=(HMI_Hour=20 AND HMI_Minute=0 AND HMI_Second=0) , Q=> );

//正极白班N清零
IF DayClear1.Q  THEN
  Par.stDT_date.An_Rectifydev_DayNG:=0;
END_IF 

IF CCD.AnRec.DayNgclassification.NgClear[1] OR DayClear1.Q  THEN
   CCD.AnRec.DayNgclassification.X1_NG :=0 ;
END_IF

IF CCD.AnRec.DayNgclassification.NgClear[2] OR DayClear1.Q  THEN
   CCD.AnRec.DayNgclassification.X2_NG :=0 ;
END_IF

IF CCD.AnRec.DayNgclassification.NgClear[3] OR DayClear1.Q  THEN
   CCD.AnRec.DayNgclassification.Y_NG :=0 ;
END_IF

IF CCD.AnRec.DayNgclassification.NgClear[4] OR DayClear1.Q  THEN
   CCD.AnRec.DayNgclassification.R_NG :=0 ;
END_IF	

IF CCD.AnRec.DayNgclassification.NgClear[5] OR DayClear1.Q  THEN
   CCD.AnRec.DayNgclassification.other_NG :=0 ;
END_IF	
	
//正极晚班NG计数
IF ((HMI_Hour>=0 AND HMI_Hour<8) OR  (HMI_Hour>=20 AND HMI_Hour<=23)) AND An_Step2>50 AND An_Step2<70  THEN
  IF CCD.AnRec.Finish.NG_Code = 1 THEN
   CCD.AnRec.NightNgclassification.X1_NG :=CCD.AnRec.NightNgclassification.X1_NG+1 ;
   CCD.AnRec.Finish.NG_Code := 0 ;
  ELSIF CCD.AnRec.Finish.NG_Code = 2 THEN
   CCD.AnRec.NightNgclassification.X2_NG := CCD.AnRec.NightNgclassification.X2_NG+1 ;  
   CCD.AnRec.Finish.NG_Code := 0 ;
  ELSIF CCD.AnRec.Finish.NG_Code = 3 THEN
   CCD.AnRec.NightNgclassification.Y_NG := CCD.AnRec.NightNgclassification.Y_NG+1 ;  
   CCD.AnRec.Finish.NG_Code := 0 ;
  ELSIF CCD.AnRec.Finish.NG_Code = 4 THEN
   CCD.AnRec.NightNgclassification.R_NG := CCD.AnRec.NightNgclassification.R_NG+1 ;   
   CCD.AnRec.Finish.NG_Code := 0 ; 
  ELSIF CCD.AnRec.Finish.NG_Code = 5 THEN 
   CCD.AnRec.NightNgclassification.other_NG :=  CCD.AnRec.NightNgclassification.other_NG+1;
   CCD.AnRec.Finish.NG_Code := 0 ;
  END_IF	
END_IF  

//正极晚班NG清零
IF  NightClear1.Q  THEN
   Par.stDT_date.An_Rectifydev_NightNG:=0;
END_IF

IF CCD.AnRec.NightNgclassification.NgClear[1] OR NightClear1.Q  THEN
   CCD.AnRec.NightNgclassification.X1_NG :=0 ;
END_IF

IF CCD.AnRec.NightNgclassification.NgClear[2] OR NightClear1.Q  THEN
   CCD.AnRec.NightNgclassification.X2_NG :=0 ;
END_IF

IF CCD.AnRec.NightNgclassification.NgClear[3] OR NightClear1.Q  THEN
   CCD.AnRec.NightNgclassification.Y_NG :=0 ;
END_IF

IF CCD.AnRec.NightNgclassification.NgClear[4] OR NightClear1.Q  THEN
   CCD.AnRec.NightNgclassification.R_NG :=0 ;
END_IF	

IF CCD.AnRec.NightNgclassification.NgClear[5] OR NightClear1.Q  THEN
   CCD.AnRec.NightNgclassification.other_NG :=0 ;
END_IF
END_ACTION

ACTION An_StandbyMain:
An_TON[1](PT:=T#0.5S);//正极拍照结果超时报警
An_TON[2](PT:=T#5S);//叠台主轴启动超时报警延时
An_TON[3](PT:=T#0.5S);
An_TON[5](PT:=T#10MS);
An_TON[6](PT:=T#0.2S);
An_TON[7](PT:=T#0.3S);
An_TON[8](PT:=T#0.3S);
An_TON[9](PT:=T#0.1S);
An_TON[10](PT:=T#2.5S);
An_TON[11](PT:=T#2.5S);
//An_StandbyStep1



IF Mach_Control.U.DT_iMode=1 THEN//在自动状态下	
	(**********************************************************************正极备料自动**********************************************************************************)
	CASE An_StandbyStep1 OF
	1000://处理负极片取 AND AN_CarryingPos1
		IF NOT DP_SinStepe THEN
			An_TON[7].IN:=TRUE;
			IF Mach_Control.An_b.An_CarryingFalg AND  Mach_Control.An_b.An_DPCarryingFalg AND  NOT Mach_Control.An_b.An_deviationFalg   AND 
			   ( CCD.AnRec.Finish.RectifyResult=1 OR Mach_Control.U.CCD_ChosesHMI	  OR Mach_Control.U.EmptyRunMode (*OR Blueflaging*)	)THEN	
					An_StandbyStep1:=6666;	//正极取料完成
			//正极搬运、叠台搬运、纠偏平台都无料---状态1
			ELSIF NOT Mach_Control.An_b.An_CarryingFalg AND  NOT Mach_Control.An_b.An_DPCarryingFalg AND NOT Mach_Control.An_b.An_deviationFalg  THEN   // 状态1  0   0    0		 	OK   				      	                             
				IF AN_CarryingPos1 THEN 
					An_StandbyStep1:=2000;//取流水线的极片	
				ELSIF AN_CarryingPos2 THEN 
					iND1:=3;
					An_StandbyStep1:=6000;//
				ELSIF (An_Step0=6666 OR An_Step0=0) AND ( An_Step3=6666 OR An_Step3=0) AND An_TON[7].Q THEN
					//Mach_Control.DT_b.Error[8]:=TRUE;//取正极片凸轮耦合时，正极取片轴不在取片位也不在叠片位报警
					An_StandbyStep1:=9993;
					AnPosError[1]:=TRUE;
				END_IF		
			//正极搬运吸盘有料，叠台搬运、纠偏台无料----状态2
			ELSIF Mach_Control.An_b.An_CarryingFalg AND  NOT Mach_Control.An_b.An_DPCarryingFalg AND  NOT Mach_Control.An_b.An_deviationFalg AND   Mach_Control.Ca_b.Ca_Quantited<>0 THEN  // 状态2  1  0  0		
				IF AN_CarryingPos1 THEN  		
					IF Mach_Control.An_b.An_deviationFPOK   THEN//需要判断热切横移轴在安全位
						DT_SingeMode();//单步选择		
						iND1:=1;	
						An_StandbyStep1:=6000;//通过凸轮耦合放极片到纠偏平台
					END_IF
				ELSIF AN_CarryingPos2  THEN			
					An_StandbyStep1:=2500;//  负极送片搬运放片到纠偏台					      					
				ELSIF (An_Step0=6666 OR An_Step0=0)  AND ( An_Step3=6666 OR An_Step3=0) AND An_TON[7].Q THEN
					//Mach_Control.DT_b.Error[8]:=TRUE;//叠负极片凸轮耦合时，负极取片轴不在耦合位报警
					An_StandbyStep1:=9993;
					AnPosError[2]:=TRUE;									   										 
				END_IF	
			//正极搬运、叠台搬运无料，纠偏台有料----状态3	
			ELSIF NOT Mach_Control.An_b.An_CarryingFalg AND  NOT Mach_Control.An_b.An_DPCarryingFalg AND  Mach_Control.An_b.An_deviationFalg THEN // 状态3    0  0  1
				IF AN_CarryingPos1 THEN  									
					IF (CCD.AnRec.Finish.RectifyResult=1 OR  Mach_Control.U.CCD_ChosesHMI OR Mach_Control.U.EmptyRunMode  (*OR  Blueflaging *))  THEN								        	
						An_TON[1].IN:=FALSE;				
						An_StandbyStep1:=2100;//取流水线的极片、同时取纠偏平台的极片
					ELSIF CCD.AnRec.Finish.RectifyResult=2 OR CCD.AnRec.Finish.RectifyResult= 3 OR CCD.AnRec.Finish.RectifyResult= 4  THEN
						//   DT_SingeMode();//单步选择			
						An_TON[1].IN:=FALSE;			
						An_StandbyStep1:=2200;//取纠偏平台的极片，再踢纠偏平台的NG片，同时取流水线的片
					ELSE
						IF NOT An_TON[1].Q THEN
							An_TON[1].IN:=TRUE;
						ELSE
							An_TON[1].IN:=FALSE;
							Mach_Control.An_b.Error[36]:=TRUE;//正极CCD第一次拍照超时
							An_StandbyStep1:=9999;
						END_IF
					END_IF
				ELSIF  AN_CarryingPos2 THEN
					IF Mach_Control.An_b.An_deviationDPOK   THEN//   
						DT_SingeMode();//单步选择		
						iND1:=2;	
						An_StandbyStep1:=6000;//通过凸轮耦合放极片到纠偏平台
					END_IF
				ELSIF (An_Step0=6666 OR An_Step0=0)  AND ( An_Step3=6666 OR An_Step3=0) AND An_TON[7].Q THEN
					//Mach_Control.DT_b.Error[8]:=TRUE;//叠负极片凸轮耦合时，负极取片轴不在耦合位报警
					 An_StandbyStep1:=9993;
					 AnPosError[3]:=TRUE;
				END_IF		
			//正极搬运吸盘有料，叠台搬运无料，纠偏台有料-----状态4
			ELSIF Mach_Control.An_b.An_CarryingFalg AND  NOT Mach_Control.An_b.An_DPCarryingFalg AND   Mach_Control.An_b.An_deviationFalg  THEN 
				IF Mach_Control.An_b.An_deviationDPOK AND arrAxisCtrl[AxiseNo.AxisName.AnDTCarryingLine].Cmd.arrbRealPoint[1]AND 
					arrAxisCtrl[AxiseNo.AxisName.AnDTCarryingLine].Status.Homed AND arrAxisCtrl[AxiseNo.AxisName.AnDTCarryingLine].Status.NoMoving
					AND (An_Step3=6666 OR An_Step3=0) THEN				
					An_StandbyStep1:=4000;//单独取纠偏平台
					An_Step3:=10;	
				END_IF
			//正极搬运吸盘无料，叠台搬运有纠偏OK料，纠偏平台无料-----状态5，流水取料且不丢NG
			ELSIF  ( Mach_Control.An_b.An_DPCarryingFalg AND  CCD.AnRec.Finish.RectifyResult=1 OR Mach_Control.U.EmptyRunMode OR  Mach_Control.U.CCD_ChosesHMI(* OR  Blueflaging*)	) AND NOT  Mach_Control.An_b.An_deviationFalg AND (An_Step0=6666 OR An_Step0=0) THEN// 状态4 正常       0 (1)     1 0    				
				IF  AN_CarryingPos1 THEN   
					IF  NOT Mach_Control.An_b.An_CarryingFalg THEN
						An_StandbyStep1:=2000;//取流水线的极片		
					END_IF
				ELSIF    An_TON[7].Q THEN// ------------------------20231209新增(An_Step0=6666 OR An_Step0=0)  AND
					  //Mach_Control.DT_b.Error[8]:=TRUE;//叠负极片凸轮耦合时，负极取片轴不在耦合位报警
					   An_StandbyStep1:=9993;
					   AnPosError[4]:=TRUE;
				END_IF			
			//	正极搬运吸盘无料，叠台搬运有纠偏NG料，纠偏台无料----状态6，取流水线极片且叠台搬运丢NG片			
			ELSIF  ( Mach_Control.An_b.An_DPCarryingFalg AND  CCD.AnRec.Finish.RectifyResult<>1 ) AND  NOT  Mach_Control.An_b.An_deviationFalg AND  NOT    Mach_Control.U.CCD_ChosesHMI AND (An_Step0=6666 OR An_Step0=0) THEN			// 状态5        0 (1)     1 0    
				   IF  AN_CarryingPos1 THEN      		
					  IF  NOT Mach_Control.an_b.An_CarryingFalg THEN    
						An_StandbyStep1:=2300;//踢纠偏平台的NG片，同时取流水线的片	     
					  ELSIF   Mach_Control.an_b.An_CarryingFalg THEN     
						An_StandbyStep1:=2400;//踢纠偏平台的NG片，同时取流水线的片	    
					  END_IF      
				   ELSIF   An_TON[7].Q THEN// ------------------------20231209新增(An_Step0=6666 OR An_Step0=0)
					  //Mach_Control.DT_b.Error[8]:=TRUE;//叠负极片凸轮耦合时，负极取片轴不在耦合位报警
					   An_StandbyStep1:=9993;
					   AnPosError[5]:=TRUE;
				  END_IF				
			END_IF	
		END_IF
	//取料流程调用				
	2000://调用取流水线子程序
		IF NOT DP_SinStepe THEN
			IF An_Step0=0 OR An_Step0=6666 THEN
				An_Step0:=10;//正极取流水线子程序
			END_IF
			DT_SingeMode();//单步选择		
			An_StandbyStep1:=2010;	
		END_IF	
	2010://判断取料是否完成
		IF An_Step0=6666 THEN
			DT_SingeMode();//单步选择		
			An_StandbyStep1:=1000;	
		END_IF				
	2100://调用取流水线子程序，取纠偏极片子程序
		IF NOT DP_SinStepe THEN
			IF An_Step0=0 OR An_Step0=6666 THEN
				An_Step0:=10;//正极取流水线子程序
			END_IF
				An_Step3:=10;//正极取纠偏平台子程序
				DT_SingeMode();//单步选择					
				An_StandbyStep1:=2110;	
		END_IF
	2110://判断正极取片流水线的极片、取纠偏平台的极片是否完成
		IF NOT DP_SinStepe THEN
			IF 	An_Step0=6666 AND 	An_Step3=6666 THEN
				DT_SingeMode();//单步选择							
				An_StandbyStep1:=1000;	
			END_IF
		END_IF			
	2200://先取纠偏平台的极片，同时根据条件判断是否可以取流水线的极片
		IF NOT DP_SinStepe THEN
			An_Step0:=10;//正极取流水线子程序
			An_Step3:=10;//正极取纠偏平台子程序
			 DT_SingeMode();//单步选择								
			An_StandbyStep1:=2210;	
		END_IF
	2210://判断取纠极片是否完成
		IF NOT DP_SinStepe THEN
			IF An_Step0=6666 AND An_Step3=6666 THEN
				An_Step2:=10;
				DT_SingeMode();//单步选择								
				An_StandbyStep1:=2220;
			END_IF
		END_IF
	2220://判断取流水线极片，踢NG极片是否完成
		IF NOT DP_SinStepe THEN
			IF   An_Step2=6666  THEN
				 DT_SingeMode();//单步选择							
				An_StandbyStep1:=1000;
			END_IF	
		END_IF
	2300://调用取流水线极片，调用踢NG片子程序
		IF NOT DP_SinStepe THEN
			An_Step0:=10;//正极取流水线子程序
			//An_Step3:=10;//正极取纠偏平台子程序
			 DT_SingeMode();//单步选择								
			An_StandbyStep1:=2310;	
		END_IF
	2310://判断取流水线极片、踢NG片是否完成
		IF NOT DP_SinStepe THEN
			IF An_Step0=6666 (*AND An_Step3=6666*) THEN
				An_Step2:=10;
				DT_SingeMode();//单步选择								
				An_StandbyStep1:=2320;
			END_IF
		END_IF
	2320:				
		IF NOT DP_SinStepe THEN
			IF   An_Step2=6666  THEN
				 DT_SingeMode();//单步选择							
				An_StandbyStep1:=1000;
			END_IF	
		END_IF			
	2400://调用踢NG片子程序
		IF NOT DP_SinStepe THEN							
			 DT_SingeMode();//单步选择								
			An_StandbyStep1:=2410;	
		END_IF
	2410://判断取流水线极片、踢NG片是否完成
		IF NOT DP_SinStepe THEN		
			An_Step2:=10;
			DT_SingeMode();//单步选择								
			An_StandbyStep1:=2420;							
		END_IF
	2420:				
		IF NOT DP_SinStepe THEN
			IF   An_Step2=6666  THEN
				DT_SingeMode();//单步选择							
				An_StandbyStep1:=1000;
			END_IF	
		END_IF			
	2500:
		IF NOT DP_SinStepe THEN
			An_Step1:=10;
			DT_SingeMode();//单步选择						
			An_StandbyStep1:=2510;	
		 END_IF
	2510:
		IF NOT DP_SinStepe THEN
			IF An_Step1=6666 THEN
				DT_SingeMode();//单步选择					
				An_StandbyStep1:=1000;
			END_IF
		END_IF									
	3030:		  // OK
		IF NOT DP_SinStepe THEN
			IF AN_CarryingPos1  THEN//正极搬运、叠片各轴在初始位
				IF CA_CarryingPos2  THEN//负极在叠片位
					IF arrAxisCtrl[AxiseNo.AxisName.SEPTATLine].Cmd.arrbRealPoint[1] THEN
						 DT_SingeMode();//单步选择	
						 IF  NOT Mach_Control.Ca_b.Ca_DPCarryingFalg  AND  Mach_Control.Ca_b.Ca_deviationFalg  AND Mach_Control.Ca_b.Ca_deviationDPOK AND TailCurlSEPTA_SafePos THEN  //叠片搬运需要取片
								 iCaCamInSel2:=1;
						  ELSE
								iCaCamInSel2:=2;
						 END_IF    
						An_StandbyStep1:=3110;//
					ELSE
						Mach_Control.DT_b.Error[6]:=TRUE;//隔膜平移不在正极片位
						An_StandbyStep1:=9991;
					END_IF
				 ELSIF  CA_CarryingPos1 THEN //负极取片位
					IF arrAxisCtrl[AxiseNo.AxisName.SEPTATLine].Cmd.arrbRealPoint[1] THEN
						  DT_SingeMode();//单步选择									
						  An_StandbyStep1:=3040;//
					ELSIF arrAxisCtrl[AxiseNo.AxisName.SEPTATLine].Cmd.arrbRealPoint[2]  THEN
							  DT_SingeMode();//单步选择			
								An_StandbyStep1:=3050;//
					ELSE
						Mach_Control.DT_b.Error[6]:=TRUE;//隔膜平移不在正极片位
						An_StandbyStep1:=9992;
					END_IF					
				ELSE
					//Mach_Control.DT_b.Error[7]:=TRUE;//叠正极片凸轮耦合时，负极取片即不在取片位，也不在叠片位
					An_StandbyStep1:=9994;
					AnPosError[7]:=TRUE;
				END_IF
			ELSE
				//Mach_Control.DT_b.Error[8]:=TRUE;//叠正极片凸轮耦合时，正极片不在取片位
				An_StandbyStep1:=9993;
				AnPosError[6]:=TRUE;
			END_IF
		END_IF		
	4000:
		IF An_Step3=6666 THEN
			An_StandbyStep1:=4100;
		END_IF
	
	4100:
		An_StandbyStep1:=1000;
	6000://判断主轴是否停止、是否在初始位、是否有轴在耦合中
		IF NOT DP_SinStepe THEN
			IF arrAxis[AxiseNo.VirAxisName.VirMain].Status.NotMoving AND arrAxis[AxiseNo.VirAxisName.VirMain].NcToPlc.SetPos=0 AND NOT DT_AxiseCoupling THEN
				DT_SingeMode();//单步选择
				An_StandbyStep1:=6024;
			ELSE
				DP_Step1:=100;//调用主轴回初始位子程序
				DT_SingeMode();//单步选择
				An_StandbyStep1:=6020;
			END_IF
		END_IF
	6020://判断主轴的模长的当前位置是否为0
		IF NOT DP_SinStepe THEN
			IF DP_Step1=6666 AND arrAxis[AxiseNo.VirAxisName.VirMain].Status.NotMoving AND arrAxis[AxiseNo.VirAxisName.VirMain].NcToPlc.SetPos=0 AND NOT DT_AxiseCoupling  THEN
				DT_SingeMode();//单步选择
				An_StandbyStep1:=6024;
			END_IF	
		END_IF	
   6024://判断NG气缸是否在安全位        无NG踢废气缸
	IF arrCyCtrl[arrCyNo.CylinderName.AnScrapbinCy].Status.ONState AND arrCyCtrl[arrCyNo.CylinderName.CaScrapbinUDCy].Status.OFFState AND
		arrCyCtrl[arrCyNo.CylinderName.CaScrapbinCy].Status.ONState AND arrCyCtrl[arrCyNo.CylinderName.PreDiaph].Status.OFFState AND 
		arrCyCtrl[arrCyNo.CylinderName.PoleHotCutterCy].Status.OFFState AND arrCyCtrl[arrCyNo.CylinderName.PoleTapeCy].Status.OFFState AND
		arrCyCtrl[arrCyNo.CylinderName.PoleTapeSplicerRCy].Status.ONState AND arrCyCtrl[arrCyNo.CylinderName.PoleTapeSplicerLCy].Status.ONState AND
        arrAxisCtrl[AxiseNo.AxisName.LeftYDUpDown].Cmd.arrbRealPoint[1] AND( arrAxisCtrl[AxiseNo.AxisName.RightYDUpDown].Cmd.arrbRealPoint[1] OR (An_OverNGMark AND arrAxisCtrl[AxiseNo.AxisName.RightYDUpDown].Cmd.arrbRealPoint[15] ))  THEN
		An_StandbyStep1:=6030;		
	ELSE
		An_StandbyStep1:=6025;	
	END_IF   
 6025:
	arrCyCtrl[arrCyNo.CylinderName.AnScrapbinCy].Cmd.bON:=TRUE;
	arrCyCtrl[arrCyNo.CylinderName.PreDiaph].Cmd.bOFF:=TRUE;
	arrCyCtrl[arrCyNo.CylinderName.PoleHotCutterCy].Cmd.bOFF:=TRUE;
	arrCyCtrl[arrCyNo.CylinderName.PoleTapeCy].Cmd.bOFF:=TRUE;
	arrCyCtrl[arrCyNo.CylinderName.PoleTapeSplicerRCy].Cmd.bON:=TRUE;
	arrCyCtrl[arrCyNo.CylinderName.PoleTapeSplicerLCy].Cmd.bON:=TRUE;
	//arrCyCtrl[arrCyNo.CylinderName.CaScrapbinCy].Cmd.bON:=TRUE;
	IF   arrCyCtrl[arrCyNo.CylinderName.AnScrapbinCy].Status.ONState AND  arrCyCtrl[arrCyNo.CylinderName.PreDiaph].Status.OFFState AND 
	arrCyCtrl[arrCyNo.CylinderName.PoleHotCutterCy].Status.OFFState AND arrCyCtrl[arrCyNo.CylinderName.PoleTapeCy].Status.OFFState AND
	arrCyCtrl[arrCyNo.CylinderName.PoleTapeSplicerRCy].Status.ONState AND arrCyCtrl[arrCyNo.CylinderName.PoleTapeSplicerLCy].Status.ONState
	AND arrCyCtrl[arrCyNo.CylinderName.CaScrapbinCy].Cmd.bON THEN
		arrCyCtrl[arrCyNo.CylinderName.CaScrapbinUDCy].Cmd.bOFF:=TRUE;		
		IF  arrCyCtrl[arrCyNo.CylinderName.CaScrapbinUDCy].Status.OFFState  AND arrAxisCtrl[AxiseNo.AxisName.LeftYDUpDown].Cmd.arrbRealPoint[1] AND
            ( arrAxisCtrl[AxiseNo.AxisName.RightYDUpDown].Cmd.arrbRealPoint[1] OR (An_OverNGMark AND arrAxisCtrl[AxiseNo.AxisName.RightYDUpDown].Cmd.arrbRealPoint[15] ))  THEN						
			An_StandbyStep1:=6024;				
		END_IF														
	END_IF  
			
	6030:						
		IF iND1=1 THEN
			An_StandbyStep1:=3030;	
		ELSIF iND1=2 THEN
			An_StandbyStep1:=3230;	
		ELSIF iND1=3 THEN
			An_StandbyStep1:=3330;			
		END_IF																												
	END_CASE
ELSE
	An_TON[1].IN:=FALSE;
	An_TON[2].IN:=FALSE;
END_IF

	
CASE An_StandbyStep1 OF
3040://负极搬运、叠片各轴在初始位，隔膜平移轴负极叠片位、正极叠片在取极片位      OK
	//正到负_正极送片搬运平 移轴凸轮耦合
	fbAnCamInCarryingLine.ParCamIn.SlaveScaling:=1;
	fbAnCamInCarryingLine.bCamInExecute:=TRUE;
	//正到负_正极送片搬运升降轴放片凸轮耦合
	fbAnCamInCarryingUpDown.iTableSel:=2;
	fbAnCamInCarryingUpDown.bCamInExecute:=TRUE;
	//正到负_正极搬运旋转轴凸轮耦合
	fbAnCamInCarryingWhirling.ParCamIn.SlaveScaling:=1;
	fbAnCamInCarryingWhirling.bCamInExecute:=TRUE;
	
	//正到负_正极叠片平移轴凸轮耦合
	fbAnCamInDTCarryingLine.ParCamIn.SlaveScaling:=1;
	fbAnCamInDTCarryingLine.bCamInExecute:=TRUE;
	
	fbAnCamInDTCarryingUpDown.iTableSel:=3;   //  //20240528SJ
    fbAnCamInDTCarryingUpDown.bCamInExecute:=TRUE;
	
	//负到正_缓存轴凸轮耦合
	fbCamInGMBuffer.iTableSel:=1;
	fbCamInGMBuffer.bCamInExecute:=TRUE;					
	//负到正_隔膜平移轴凸轮耦合
	fbCamInGMDanserMove.iTableSel:=1;
	fbCamInGMDanserMove.bCamInExecute:=TRUE;
	//隔膜驱动
	fbCamInVirGMDriver.iTableSel:=1;
	fbCamInVirGMDriver.bCamInExecute:=TRUE;		
																
	//I判断凸轮耦合是否完成
		IF fbAnCamInCarryingLine.bInSync AND fbAnCamInCarryingUpDown.bInSync AND fbAnCamInCarryingWhirling.bInSync AND
			fbAnCamInDTCarryingLine.bInSync AND  fbAnCamInDTCarryingUpDown.bInSync AND ////  //20240528SJ
			 fbCamInGMBuffer.bInSync AND fbCamInGMDanserMove.bInSync  AND  fbCamInVirGMDriver.bInSync    THEN 
			DT_SingeMode();//单步选择	
			An_StandbyStep1:=3060;
		ELSIF fbAnCamInCarryingLine.bError OR fbAnCamInCarryingUpDown.bError OR fbAnCamInCarryingWhirling.bError OR
			fbAnCamInDTCarryingLine.bError OR 
			 fbCamInGMBuffer.bError OR fbCamInGMDanserMove.bError  OR  fbCamInVirGMDriver.bError  THEN 	   
			Mach_Control.DT_b.Error[19]:=TRUE;//凸轮耦合报警
			An_StandbyStep1:=9995;
		END_IF		

		3060://主轴启动    OK					  
			IF fbAnCamInCarryingLine.bInSync AND fbAnCamInCarryingUpDown.bInSync AND fbAnCamInCarryingWhirling.bInSync AND
				fbAnCamInDTCarryingLine.bInSync AND  fbCamInGMBuffer.bInSync AND  fbCamInGMDanserMove.bInSync  AND
				fbCamInVirGMDriver.bInSync    AND
				AN_CarryingPos1 AND  CA_CarryingPos1 AND  arrAxisCtrl[AxiseNo.AxisName.SEPTATLine].Cmd.arrbRealPoint[1] THEN
				arrAxisCtrl[AxiseNo.VirAxisName.VirMain].Cmd	.bDynamitcsParSel:=2;	
				arrAxisPar[AxiseNo.VirAxisName.VirMain].fTagatTime:=VirMain_TagatTime;
				arrAxisCtrl[AxiseNo.VirAxisName.VirMain].Cmd	.fPositon_of_Abs:=360;
				arrAxisCtrl[AxiseNo.VirAxisName.VirMain].Cmd	.bMoveAbs:=TRUE;	
			END_IF			
			
			IF  arrAxis[AxiseNo.VirAxisName.VirMain].Status.Moving OR arrAxisCtrl[AxiseNo.VirAxisName.VirMain].Status.fActPos>=10  THEN
				arrAxisCtrl[AxiseNo.VirAxisName.VirMain].Cmd	.bMoveAbs:=FALSE;	
				An_TON[2].IN:=FALSE;			
				An_StandbyStep1:=3070;
				An_StandbyStep2:=100;	//判断真空、破真空
				An_StandbyStep3:=100;
				DP_Step8:=200;//纠偏平台有无极片复检
			ELSE
				IF NOT An_TON[2].Q THEN
					An_TON[2].IN:=TRUE;
				ELSE
					An_TON[2].IN:=FALSE;
					Mach_Control.DT_b.Error[22]:=TRUE;//主轴启动超时报警
					arrAxisCtrl[AxiseNo.VirAxisName.VirMain].Cmd	.bMoveAbs:=FALSE;
					An_StandbyStep1:=10000;	
				END_IF
			END_IF	


		3050://负极搬运、叠片各轴在初始位，隔膜平移轴正极叠片位、正极叠片在取极片位    OK
						//正到负_正极送片搬运平移轴凸轮耦合
							fbAnCamInCarryingLine.ParCamIn.SlaveScaling:=1;
							fbAnCamInCarryingLine.bCamInExecute:=TRUE;						
						//正到负_正极送片搬运升降轴放片凸轮耦合
							fbAnCamInCarryingUpDown.iTableSel:=2;
							fbAnCamInCarryingUpDown.bCamInExecute:=TRUE;
						//正到负_正极叠片平移轴凸轮耦合
							fbAnCamInDTCarryingLine.ParCamIn.SlaveScaling:=1;
							fbAnCamInDTCarryingLine.bCamInExecute:=TRUE;		
							
							fbAnCamInDTCarryingUpDown.iTableSel:=3;   //  //20240528SJ
							fbAnCamInDTCarryingUpDown.bCamInExecute:=TRUE;
			
						//正到负_正极搬运旋转轴凸轮耦合		
							fbAnCamInCarryingWhirling.ParCamIn.SlaveScaling:=1;
							fbAnCamInCarryingWhirling.bCamInExecute:=TRUE;								 
						//判断凸轮耦合是否完成
							IF fbAnCamInCarryingLine.bInSync AND fbAnCamInCarryingUpDown.bInSync   AND fbAnCamInCarryingWhirling.bInSync AND
                                  fbAnCamInDTCarryingLine.bInSync   AND   fbAnCamInDTCarryingUpDown.bInSync         THEN
			                        DT_SingeMode();//单步选择		
								    An_StandbyStep1:=3080;
							ELSIF fbAnCamInCarryingLine.bError OR  fbAnCamInCarryingUpDown.bError  OR fbAnCamInCarryingWhirling.bError  OR 
                                     fbAnCamInDTCarryingLine.bError   OR  fbAnCamInDTCarryingUpDown.bError     THEN
								Mach_Control.DT_b.Error[19]:=TRUE;//凸轮耦合报警
								An_StandbyStep1:=9996;								
							END_IF				
		3080://主轴启动    OK					  
			IF fbAnCamInCarryingLine.bInSync AND fbAnCamInCarryingUpDown.bInSync   AND fbAnCamInCarryingWhirling.bInSync AND
                  		fbAnCamInDTCarryingLine.bInSync  AND
 				  AN_CarryingPos1 AND  CA_CarryingPos1 AND  arrAxisCtrl[AxiseNo.AxisName.SEPTATLine].Cmd.arrbRealPoint[2] THEN
				arrAxisCtrl[AxiseNo.VirAxisName.VirMain].Cmd	.bDynamitcsParSel:=2;	
				arrAxisPar[AxiseNo.VirAxisName.VirMain].fTagatTime:=VirMain_TagatTime;
				arrAxisCtrl[AxiseNo.VirAxisName.VirMain].Cmd	.fPositon_of_Abs:=360;
				arrAxisCtrl[AxiseNo.VirAxisName.VirMain].Cmd	.bMoveAbs:=TRUE;	
			END_IF			
			
			IF  arrAxis[AxiseNo.VirAxisName.VirMain].Status.Moving OR arrAxisCtrl[AxiseNo.VirAxisName.VirMain].Status.fActPos>=10  THEN
						arrAxisCtrl[AxiseNo.VirAxisName.VirMain].Cmd	.bMoveAbs:=FALSE;	
						An_TON[2].IN:=FALSE;			
						An_StandbyStep1:=3090;
						An_StandbyStep2:=100;	//判断真空、破真空
						An_StandbyStep3:=100;
						DP_Step8:=200;//纠偏平台有无极片复检
			ELSE
						IF NOT An_TON[2].Q THEN
							An_TON[2].IN:=TRUE;
						ELSE
							An_TON[2].IN:=FALSE;
							Mach_Control.DT_b.Error[22]:=TRUE;//主轴启动超时报警
							arrAxisCtrl[AxiseNo.VirAxisName.VirMain].Cmd	.bMoveAbs:=FALSE;
							An_StandbyStep1:=10000;	
						END_IF
			END_IF	
	

		3110://负极搬运、叠片各轴在初始位，隔膜平移轴负极叠片位、正极叠片在放极片初始位       OK
						//正到负_正极送片搬运平移轴凸轮耦合
							fbAnCamInCarryingLine.ParCamIn.SlaveScaling:=1;
							fbAnCamInCarryingLine.bCamInExecute:=TRUE;	
						//正到负_正极送片搬运升降轴放片凸轮耦合
							fbAnCamInCarryingUpDown.iTableSel:=2;
							fbAnCamInCarryingUpDown.bCamInExecute:=TRUE;
						//正到负_正极搬运旋转轴凸轮耦合		
							fbAnCamInCarryingWhirling.ParCamIn.SlaveScaling:=1;
							fbAnCamInCarryingWhirling.bCamInExecute:=TRUE;		
							
						//正到负_正极叠片平移轴凸轮耦合
							fbAnCamInDTCarryingLine.ParCamIn.SlaveScaling:=1;
							fbAnCamInDTCarryingLine.bCamInExecute:=TRUE;	

							fbAnCamInDTCarryingUpDown.iTableSel:=3;   //  //20240528SJ
                            fbAnCamInDTCarryingUpDown.bCamInExecute:=TRUE;
												
						//正到负_负极送片搬运平移轴凸轮耦合
							fbCaCamInCarryingLine2.ParCamIn.SlaveScaling:=-1;
							fbCaCamInCarryingLine2.bCamInExecute:=TRUE;
							fbCaCamInCarryingUpDown2.iTableSel:=3; //20240528SJ
                            fbCaCamInCarryingUpDown2.bCamInExecute:=TRUE;
							
							
					 IF  	iCaCamInSel1=1 THEN	
						//正到负_负极送片搬运升降轴取片凸轮耦合 
					//		fbCaCamInCarryingUpDown2.iTableSel:=1;
					//		 fbCaCamInCarryingUpDown2.bCamInExecute:=TRUE;
					 END_IF
		 
						//正到负_负极叠片搬运平移轴凸轮耦合
							fbCaCamInDTCarryingLine.ParCamIn.SlaveScaling:=-1;
							fbCaCamInDTCarryingLine.bCamInExecute:=TRUE;
					 IF  	iCaCamInSel2=1 THEN			
						//正到负_负极叠片搬运升降轴取片凸轮耦合
							fbCaCamInDTCarryingUpDown.iTableSel:=1;
							fbCaCamInDTCarryingUpDown.bCamInExecute:=TRUE;
					ELSE
							fbCaCamInDTCarryingUpDown.iTableSel:=3;   //20240528SJ
							fbCaCamInDTCarryingUpDown.bCamInExecute:=TRUE;		
				     END_IF	
						
					
									//负到正_缓存轴凸轮耦合
							fbCamInGMBuffer.iTableSel:=1;
							fbCamInGMBuffer.bCamInExecute:=TRUE;					
						//负到正_隔膜平移轴凸轮耦合
							fbCamInGMDanserMove.iTableSel:=1;
							fbCamInGMDanserMove.bCamInExecute:=TRUE;
                       //隔膜驱动
							fbCamInVirGMDriver.iTableSel:=1;
						    fbCamInVirGMDriver.bCamInExecute:=TRUE;				
							
				
						//判断凸轮是否耦合完成
							IF fbAnCamInCarryingLine.bInSync AND fbAnCamInCarryingUpDown.bInSync AND  fbAnCamInCarryingWhirling.bInSync AND
                                fbAnCamInDTCarryingLine.bInSync AND   fbAnCamInDTCarryingUpDown.bInSync AND 
							   	fbCaCamInCarryingLine2.bInSync      AND   fbCaCamInCarryingUpDown2.bInSync    AND   // (  (fbCaCamInCarryingUpDown2.bInSync AND iCaCamInSel1=1) OR       iCaCamInSel1=2 ) 
							 	fbCaCamInDTCarryingLine.bInSync AND  (  (fbCaCamInDTCarryingUpDown.bInSync   AND iCaCamInSel2=1)  OR  (  iCaCamInSel2=2  AND fbCaCamInDTCarryingUpDown.bInSync )   )    AND
                                fbCamInGMBuffer.bInSync AND  fbCamInGMDanserMove.bInSync  AND  fbCamInVirGMDriver.bInSync  THEN
 
										IF Mach_Control.DT_b.SinStepMode THEN//单步调试模式
											DP_SinStepe:=TRUE;
										ELSE
											DP_SinStepe:=FALSE;	
										END_IF
										An_StandbyStep1:=3120;	
							ELSIF fbAnCamInCarryingLine.bError OR fbAnCamInCarryingUpDown.bError OR  fbAnCamInCarryingWhirling.bError OR
                                fbAnCamInDTCarryingLine.bError OR fbAnCamInDTCarryingUpDown.bError OR
							     fbCaCamInCarryingLine2.bError   OR fbCaCamInCarryingUpDown2.bError     OR
							 	 fbCaCamInDTCarryingLine.bError OR fbCaCamInDTCarryingUpDown.bError   OR
                                 fbCamInGMBuffer.bError OR  fbCamInGMDanserMove.bError  OR  fbCamInVirGMDriver.bError  THEN
									Mach_Control.DT_b.Error[19]:=TRUE;//凸轮耦合报警
									An_StandbyStep1:=9997;	
							END_IF
	3120://主轴启动		
			IF fbAnCamInCarryingLine.bInSync AND fbAnCamInCarryingUpDown.bInSync AND  fbAnCamInCarryingWhirling.bInSync AND
				fbAnCamInDTCarryingLine.bInSync AND fbCaCamInCarryingLine2.bInSync    AND
			     // (  (fbCaCamInCarryingUpDown2.bInSync AND iCaCamInSel1=1) OR       iCaCamInSel1=2 )     AND
				fbCaCamInDTCarryingLine.bInSync AND  (  (fbCaCamInDTCarryingUpDown.bInSync   AND iCaCamInSel2=1)  OR  iCaCamInSel2=2 )    AND
				 fbCamInGMBuffer.bInSync AND  fbCamInGMDanserMove.bInSync  AND  fbCamInVirGMDriver.bInSync  AND
 				AN_CarryingPos1 AND  CA_CarryingPos2 AND  arrAxisCtrl[AxiseNo.AxisName.SEPTATLine].Cmd.arrbRealPoint[1] THEN
						arrAxisCtrl[AxiseNo.VirAxisName.VirMain].Cmd	.bDynamitcsParSel:=2;	
						arrAxisPar[AxiseNo.VirAxisName.VirMain].fTagatTime:=VirMain_TagatTime;
						arrAxisCtrl[AxiseNo.VirAxisName.VirMain].Cmd	.fPositon_of_Abs:=360;
						arrAxisCtrl[AxiseNo.VirAxisName.VirMain].Cmd	.bMoveAbs:=TRUE;	
		    END_IF				
			
			IF  arrAxis[AxiseNo.VirAxisName.VirMain].Status.Moving OR arrAxisCtrl[AxiseNo.VirAxisName.VirMain].Status.fActPos>=10 THEN
						arrAxisCtrl[AxiseNo.VirAxisName.VirMain].Cmd	.bMoveAbs:=FALSE;	
						An_TON[2].IN:=FALSE;	
						An_StandbyStep1:=3130;
						An_StandbyStep2:=200;
						An_StandbyStep3:=200;
						DP_Step8:=200;//纠偏平台有无极片复检
			ELSE
						IF NOT An_TON[2].Q THEN
							An_TON[2].IN:=TRUE;
						ELSE
							An_TON[2].IN:=FALSE;
							Mach_Control.DT_b.Error[22]:=TRUE;//主轴启动超时报警
							arrAxisCtrl[AxiseNo.VirAxisName.VirMain].Cmd	.bMoveAbs:=FALSE;	
							An_StandbyStep1:=10000;	
						END_IF
			END_IF
	
	3230	:				//OK			
		//正极送片搬运平移
		fbAnCamInCarryingLine.ParCamIn.SlaveScaling:=-1;
		fbAnCamInCarryingLine.bCamInExecute:=TRUE;						
		//正极送片搬运升降
		fbAnCamInCarryingUpDown.iTableSel:=3;       //20240528SJ  
		fbAnCamInCarryingUpDown.bCamInExecute:=TRUE;		
		//正极送片搬运旋转
		fbAnCamInCarryingWhirling.ParCamIn.SlaveScaling:=-1;
		fbAnCamInCarryingWhirling.bCamInExecute:=TRUE;		
						
		//正极叠台搬运平移
		fbAnCamInDTCarryingLine.ParCamIn.SlaveScaling:=-1;
		fbAnCamInDTCarryingLine.bCamInExecute:=TRUE;	
		//正极叠片搬运升降
		fbAnCamInDTCarryingUpDown.iTableSel:=1;       //    
		fbAnCamInDTCarryingUpDown.bCamInExecute:=TRUE;		
	
	
		  IF fbAnCamInCarryingLine.bInSync AND fbAnCamInCarryingWhirling.bInSync AND   fbAnCamInCarryingUpDown.bInSync AND
				fbAnCamInDTCarryingLine.bInSync   AND  fbAnCamInDTCarryingUpDown.bInSync   THEN 
				  DT_SingeMode();//单步选择		
				  An_StandbyStep1:=3240;
		 ELSIF fbAnCamInCarryingLine.bError OR fbAnCamInCarryingWhirling.bError OR  fbAnCamInCarryingUpDown.bError OR
				fbAnCamInDTCarryingLine.bError   OR  fbAnCamInDTCarryingUpDown.bError   THEN 
					 Mach_Control.DT_b.Error[19]:=TRUE;//凸轮耦合报警
					 An_StandbyStep1:=9998;
		END_IF	 

	3240:					//OK	
				IF fbAnCamInCarryingLine.bInSync AND fbAnCamInCarryingWhirling.bInSync AND
					fbAnCamInDTCarryingLine.bInSync   AND  fbAnCamInDTCarryingUpDown.bInSync  AND AN_CarryingPos2  THEN 	
					  arrAxisCtrl[AxiseNo.VirAxisName.VirMain].Cmd	.bDynamitcsParSel:=2;	
					  arrAxisPar[AxiseNo.VirAxisName.VirMain].fTagatTime:=VirMain_TagatTime;
					  arrAxisCtrl[AxiseNo.VirAxisName.VirMain].Cmd	.fPositon_of_Abs:=360;
					  arrAxisCtrl[AxiseNo.VirAxisName.VirMain].Cmd	.bMoveAbs:=TRUE;				
				END_IF	
	
				IF  arrAxis[AxiseNo.VirAxisName.VirMain].Status.Moving AND arrAxisCtrl[AxiseNo.VirAxisName.VirMain].Status.fModuloActPos>=5  THEN		
						arrAxisCtrl[AxiseNo.VirAxisName.VirMain].Cmd	.bMoveAbs:=FALSE;
						An_TON[2].IN:=FALSE;		
						An_StandbyStep1:=3250;	
						An_StandbyStep2:=300;//正极取极片
						An_StandbyStep3:=300;
				ELSE
						IF NOT An_TON[2].Q THEN
							An_TON[2].IN:=TRUE;
						ELSE
					 	An_TON[2].IN:=FALSE;
							Mach_Control.DT_b.Error[22]:=TRUE;//主轴启动超时报警
							arrAxisCtrl[AxiseNo.VirAxisName.VirMain].Cmd	.bMoveAbs:=FALSE;	
							An_StandbyStep1:=10000;	
						END_IF
			  END_IF

	3330:		//OK	
		//正极送片搬运平移
			fbAnCamInCarryingLine.ParCamIn.SlaveScaling:=-1;
			fbAnCamInCarryingLine.bCamInExecute:=TRUE;							
		//正极送片搬运升降取片
		  fbAnCamInCarryingUpDown.iTableSel:=3;       //20240528SJ   
		  fbAnCamInCarryingUpDown.bCamInExecute:=TRUE;			
		
		//正极叠台搬运平移
				fbAnCamInDTCarryingLine.ParCamIn.SlaveScaling:=-1;
				fbAnCamInDTCarryingLine.bCamInExecute:=TRUE;	
				fbAnCamInDTCarryingUpDown.iTableSel:=3;   //  //20240528SJ
                fbAnCamInDTCarryingUpDown.bCamInExecute:=TRUE;
					
		//	正极送片搬运旋转
			fbAnCamInCarryingWhirling.ParCamIn.SlaveScaling:=-1;
			fbAnCamInCarryingWhirling.bCamInExecute:=TRUE;		
					
		IF fbAnCamInCarryingLine.bInSync AND  fbAnCamInCarryingUpDown.bInSync AND
			fbAnCamInDTCarryingLine.bInSync   AND fbAnCamInCarryingWhirling.bInSync AND  fbAnCamInDTCarryingUpDown.bInSync   THEN   
			  DT_SingeMode();//单步选择		
			  An_StandbyStep1:=3340;
		ELSIF fbAnCamInCarryingLine.bError  OR  fbAnCamInCarryingUpDown.bError OR 
			fbAnCamInDTCarryingLine.bError  OR fbAnCamInCarryingWhirling.bError  OR   fbAnCamInDTCarryingUpDown.bError  THEN   
				 Mach_Control.DT_b.Error[29]:=TRUE;//凸轮耦合报警
				 An_StandbyStep1:=9998;
		END_IF	 	

	3340:  //OK
				IF fbAnCamInCarryingLine.bInSync AND fbAnCamInDTCarryingLine.bInSync   AND fbAnCamInCarryingWhirling.bInSync  AND 
					 AN_CarryingPos2  THEN   
					  arrAxisCtrl[AxiseNo.VirAxisName.VirMain].Cmd	.bDynamitcsParSel:=2;	
					  arrAxisPar[AxiseNo.VirAxisName.VirMain].fTagatTime:=VirMain_TagatTime;
					  arrAxisCtrl[AxiseNo.VirAxisName.VirMain].Cmd	.fPositon_of_Abs:=360;
					  arrAxisCtrl[AxiseNo.VirAxisName.VirMain].Cmd	.bMoveAbs:=TRUE;	
				END_IF	 			
				
				IF  arrAxis[AxiseNo.VirAxisName.VirMain].Status.Moving OR arrAxisCtrl[AxiseNo.VirAxisName.VirMain].Status.fActPos>=5  THEN		
						arrAxisCtrl[AxiseNo.VirAxisName.VirMain].Cmd	.bMoveAbs:=FALSE;
							An_TON[2].IN:=FALSE;
							An_StandbyStep1:=3350;
							An_StandbyStep2:=400;//						
							An_StandbyStep3:=400;//正极主分料皮带清零
				ELSE
						IF NOT An_TON[2].Q THEN
						    An_TON[2].IN:=TRUE;
						ELSE
						An_TON[2].IN:=FALSE;
						Mach_Control.DT_b.Error[22]:=TRUE;//主轴启动超时报警
						arrAxisCtrl[AxiseNo.VirAxisName.VirMain].Cmd	.bMoveAbs:=FALSE;	
						An_StandbyStep1:=10000;	
					END_IF
			  END_IF				
END_CASE
END_ACTION

ACTION An_StandbyMain2:

//An_StandbyStep2-------真空处理
//An_StandbyStep3-------主轴位置判断

CASE An_StandbyStep2 OF
100://正极叠片     负极在取片位
       bStandbyStep1_3:=FALSE;
       bStandbyStep1_4:=FALSE;
       An_StandbyStep2:=110; 
	   
110:
	IF arrAxisCtrl[AxiseNo.VirAxisName.VirMain].Status.fActPos>=20  AND  arrAxisCtrl[AxiseNo.VirAxisName.VirMain].Status.fActPos<=30     THEN
	//正送片搬运极取片处理
		IF   arrAxisCtrl[AxiseNo.AxisName.CaCarryingUpDown2].Cmd.arrbRealPoint[4] AND 
		      NOT Mach_Control.Ca_b.Ca_CarryingFalg    AND  ( Mach_Control.Ca_b.Ca_CacheBeltDLOK OR  Mach_Control.U.EmptyRunMode )  AND 
		      NOT  Mach_Control.Ca_b.Ca_CacheBelting   AND NOT  bStandbyStep1_3  THEN
			   Ca_Step0:=10;//负极取流水线子程序
			   bStandbyStep1_3:=TRUE;
		END_IF
					
		IF arrAxisCtrl[AxiseNo.AxisName.CaDTCarryingUpDown].Cmd.arrbRealPoint[4] AND 
			NOT Mach_Control.Ca_b.Ca_DPCarryingFalg AND   Mach_Control.Ca_b.Ca_deviationFalg AND  ( CCD.CaRec.Finish.RectifyResult=1 OR Mach_Control.U.EmptyRunMode  )  AND 
			NOT  bStandbyStep1_4   THEN
			Ca_Step3:=10;//正极取纠偏平台子程序
			bStandbyStep1_4:=TRUE;
		END_IF
		 
	ELSIF  arrAxisCtrl[AxiseNo.VirAxisName.VirMain].Status.fActPos>245  THEN
		An_StandbyStep2:=120;
	END_IF
		
120:	
	IF 	arrAxisCtrl[AxiseNo.VirAxisName.VirMain].Status.fActPos>=260  AND   arrAxisCtrl[AxiseNo.VirAxisName.VirMain].Status.fActPos<=320   THEN//198
			arrCyCtrl[arrCyNo.ElectValveName.AnCarryingVacuum].Cmd.bON:=FALSE;////搬运真空破真空				
			arrCyCtrl[arrCyNo.ElectValveName.AnCarryingVacuum].Cmd.bOFF:=TRUE;////搬运真空破真空		

			arrCyCtrl[arrCyNo.ElectValveName.AnCarryingVacuumBark].Cmd.bON:=TRUE;////搬运真空破真空				
			arrCyCtrl[arrCyNo.ElectValveName.AnCarryingVacuumBark].Cmd.bOFF:=FALSE;////搬运真空破真空
			arrCyCtrl[arrCyNo.ElectValveName.AndeviationVacuum].Cmd.bON:=TRUE;//纠偏平台开真空
			arrCyCtrl[arrCyNo.ElectValveName.AndeviationVacuum].Cmd.bOFF:=FALSE;//纠偏平台开真空
			//IF Mach_Control.An_b.An_CarryingFalg THEN
				Mach_Control.An_b.An_deviationFalg:=TRUE;//置位纠偏平台上有料标记
				Mach_Control.An_b.An_CarryingFalg :=FALSE;//复位正极搬运机械手有料标记
			//END_IF
			Par.stDT_date.An_MQ_Slice[1]:=Par.stDT_date.An_MQ_Slice[0];
			An_StandbyStep2:=6666;
	END_IF	
					
				
 200:	     // 状态2         1         0       0     iMD1:=1;	  	Ca_StandbyStep0:=6000;//通过凸轮耦合放极片到纠偏平台
	 IF arrAxisCtrl[AxiseNo.VirAxisName.VirMain].Status.fActPos>=CamOutArgel+15 THEN   //整机叠片搬运
			 IF iCaCamInSel2=1  THEN	 
				 arrCyCtrl[arrCyNo.ElectValveName.CaDTCarryingVacuum].Cmd.bON:=FALSE;//负极叠片搬运真空开
				arrCyCtrl[arrCyNo.ElectValveName.CaDTCarryingVacuum].Cmd.bOFF:=TRUE;//负极叠片搬运真空开
			 END_IF
			An_StandbyStep2:=205;
	 END_IF
205:
	 IF arrAxisCtrl[AxiseNo.VirAxisName.VirMain].Status.fActPos>=235 THEN   //整机叠片搬运
			IF Mach_Control.DT_b.DT_CCD_TwoModel  AND iCaCamInSel2=1    THEN												
				CCD.CaRec.Finish.RectifyResult:=0;
				CCD.CaRec.Finish.RectifyX1:=0;
				CCD.CaRec.Finish.RectifyX2:=0;
				CCD.CaRec.Finish.RectifyY:=0;												
				Mach_Control.Ca_b.Ca_CCDStart :=TRUE;//启动CCD拍照
				CCD.CaRec.Start.iPhotoDo:=2;//第二次拍照
				CCD.CaRec.Start.stPoleNo:=Par.stDT_date.Ca_MQ_Slice[8].stPoleNo;  //???????????????????????????
			END_IF
			An_StandbyStep2:=210;
	END_IF 
 210:
	IF arrAxisCtrl[AxiseNo.VirAxisName.VirMain].Status.fActPos>=250  AND arrAxisCtrl[AxiseNo.VirAxisName.VirMain].Status.fActPos<=(250+6) AND NOT Mach_Control.Ca_b.Ca_CacheBelting THEN
		//IF iCaCamInSel1=1  THEN   //  正极送片搬运  
			IF ( Mach_Control.Ca_b.Ca_CacheBeltDLOK  OR  Mach_Control.U.EmptyRunMode )     AND   NOT Mach_Control.Ca_b.Ca_CarryingFalg  THEN
				Ca_Step0:=10;  //调用升降取片流程 
			ELSE
				IF NOT Mach_Control.Ca_b.Ca_CarryingFalg THEN
					//fbAnCamInCarryingUpDown.bCamInExecute:=FALSE;//正极升解除耦合
					Mach_Control.Ca_b.Ca_CacheBelting:=FALSE;//正极搬运升降取极片中	
					arrCyCtrl[arrCyNo.ElectValveName.CaCarryingVacuum2].Cmd.bON:=FALSE;	//负极送片搬运升降真空									
					arrCyCtrl[arrCyNo.ElectValveName.CaCarryingVacuum2].Cmd.bOFF:=TRUE;	//负极送片搬运升降真空			
				END_IF																									
				IF NOT arrAxisCtrl[AxiseNo.AxisName.CaCarryingUpDown2].Cmd.arrbRealPoint[4] THEN
					arrAxisCtrl[AxiseNo.AxisName.CaCarryingUpDown2].Cmd.iGoSetPos:=4;//移动至流水线上方
				END_IF	
			END_IF	
		//ELSE	    		
		//		;
		//END_IF			
	An_StandbyStep2:=220;
	END_IF
				
  220:			
	IF 	arrAxisCtrl[AxiseNo.VirAxisName.VirMain].Status.fActPos>=260   AND  arrAxisCtrl[AxiseNo.VirAxisName.VirMain].Status.fActPos<=320  THEN//198
		arrCyCtrl[arrCyNo.ElectValveName.AnCarryingVacuum].Cmd.bON:=FALSE;////搬运真空破真空				
		arrCyCtrl[arrCyNo.ElectValveName.AnCarryingVacuum].Cmd.bOFF:=TRUE;////搬运真空破真空
		arrCyCtrl[arrCyNo.ElectValveName.AnCarryingVacuumBark].Cmd.bON:=TRUE;////搬运真空破真空				
		arrCyCtrl[arrCyNo.ElectValveName.AnCarryingVacuumBark].Cmd.bOFF:=FALSE;////搬运真空破真空
		arrCyCtrl[arrCyNo.ElectValveName.AndeviationVacuum].Cmd.bON:=TRUE;//纠偏平台开真空
		arrCyCtrl[arrCyNo.ElectValveName.AndeviationVacuum].Cmd.bOFF:=FALSE;//纠偏平台开真空
		//IF Mach_Control.An_b.An_CarryingFalg THEN
			Mach_Control.An_b.An_deviationFalg:=TRUE;//置位纠偏平台上有料标记
			Mach_Control.An_b.An_CarryingFalg:=FALSE;//复位负极送片搬运吸盘上有料标记			
		//END_IF
		Par.stDT_date.An_MQ_Slice[1]:=Par.stDT_date.An_MQ_Slice[0];
	
		IF 	 iCaCamInSel2=1  THEN
			arrCyCtrl[arrCyNo.ElectValveName.CaDTCarryingVacuum].Cmd.bON:=FALSE;	//负极叠台搬运升降真空开	
			arrCyCtrl[arrCyNo.ElectValveName.CaDTCarryingVacuum].Cmd.bOFF:=TRUE;	//负极叠台搬运升降真空开	
			arrCyCtrl[arrCyNo.ElectValveName.CadeviationVacuum].Cmd.bON:=FALSE;	//负极纠偏台真空破真空			
			arrCyCtrl[arrCyNo.ElectValveName.CadeviationVacuum].Cmd.bOFF:=TRUE;	//负极纠偏台真空破真空											
			arrCyCtrl[arrCyNo.ElectValveName.CadeviationVacuumBark].Cmd.bON:=TRUE;	//负极纠偏台真空破真空			
			arrCyCtrl[arrCyNo.ElectValveName.CadeviationVacuumBark].Cmd.bOFF:=FALSE;	//负极纠偏台真空破真空	
			//IF Mach_Control.Ca_b.Ca_deviationFalg THEN		
				Mach_Control.Ca_b.Ca_DPCarryingFalg :=TRUE;//正极叠片搬运吸盘上有料标记
				Mach_Control.Ca_b.Ca_deviationFalg:=FALSE;//置位纠偏平台上有料标记
			//END_IF
			Par.stDT_date.Ca_MQ_Slice[9]:=Par.stDT_date.Ca_MQ_Slice[8];
		ELSE
			;
		END_IF	
	An_StandbyStep2:=666;
	END_IF			

300:	     // 状态2         1         0       0     iMD1:=1;	  	Ca_StandbyStep0:=6000;//通过凸轮耦合放极片到纠偏平台
 			 IF arrAxisCtrl[AxiseNo.VirAxisName.VirMain].Status.fActPos>=CamOutArgel+15 THEN   //整机叠片搬运
						arrCyCtrl[arrCyNo.ElectValveName.AnDTCarryingVacuum].Cmd.bON:=FALSE;//正极叠片搬运真空
						arrCyCtrl[arrCyNo.ElectValveName.AnDTCarryingVacuum].Cmd.bOFF:=TRUE;//正极叠片搬运真空
			    An_StandbyStep2:=305;
			 END_IF
305:
			IF arrAxisCtrl[AxiseNo.VirAxisName.VirMain].Status.fActPos>=235 THEN
				    //	正极送片搬运			在子流程中处理								
					IF Mach_Control.DT_b.DT_CCD_TwoModel     THEN												
						CCD.AnRec.Finish.RectifyResult:=0;
						CCD.AnRec.Finish.RectifyX1:=0;
						CCD.AnRec.Finish.RectifyX2:=0;
						CCD.AnRec.Finish.RectifyY:=0;												
						Mach_Control.An_b.An_CCDStart :=TRUE;//启动CCD拍照
						CCD.AnRec.Start.iPhotoDo:=2;//第二次拍照
						CCD.CaRec.Start.stPoleNo:=Par.stDT_date.Ca_MQ_Slice[8].stPoleNo;  //???????????????????????????
					END_IF	
					 An_StandbyStep2:=310;
			END_IF		 
 310:
				IF arrAxisCtrl[AxiseNo.VirAxisName.VirMain].Status.fActPos>=250  AND arrAxisCtrl[AxiseNo.VirAxisName.VirMain].Status.fActPos<=(250+6) AND NOT Mach_Control.An_b.An_MainBelting THEN
							 IF (Mach_Control.An_b.An_MainBeltOK  OR  Mach_Control.U.EmptyRunMode )  AND  NOT Mach_Control.An_b.An_CarryingFalg (*AND NOT Mach_Control.An_b.JumpPiceReady*)  THEN
								//fbAnCarryingVacuum.Vacuumsel:=1;										
								// Mach_Control.An_b.An_MainBelting:=TRUE;//正极搬运升降取极片中	 
								An_Step0:=10;  //调用升降取片流程 
							 ELSE
									//fbAnCamInCarryingUpDown.bCamInExecute:=FALSE;//正极升解除耦合
									Mach_Control.An_b.An_MainBelting:=FALSE;//正极搬运升降取极片中	
									arrCyCtrl[arrCyNo.ElectValveName.AnCarryingVacuumBark].Cmd.bON:=FALSE;////搬运真空破真空				
									arrCyCtrl[arrCyNo.ElectValveName.AnCarryingVacuumBark].Cmd.bOFF:=FALSE;////搬运真空破真空
									arrCyCtrl[arrCyNo.ElectValveName.AnCarryingVacuum].Cmd.bON:=FALSE;////搬运真空破真空				
									arrCyCtrl[arrCyNo.ElectValveName.AnCarryingVacuum].Cmd.bOFF:=FALSE;////搬运真空破真空									
									IF NOT arrAxisCtrl[AxiseNo.AxisName.AnCarryingUpDown].Cmd.arrbRealPoint[4] THEN
										arrAxisCtrl[AxiseNo.AxisName.AnCarryingUpDown].Cmd.iGoSetPos:=4;//移动至流水线上方
									END_IF	
							END_IF	
				          An_StandbyStep2:=320;
				END_IF
				
320:			
			IF 	arrAxisCtrl[AxiseNo.VirAxisName.VirMain].Status.fActPos>=260    AND    	arrAxisCtrl[AxiseNo.VirAxisName.VirMain].Status.fActPos<=320  THEN//198
					//正极送片搬运
						arrCyCtrl[arrCyNo.ElectValveName.AnDTCarryingVacuum].Cmd.bON:=FALSE;//叠台搬运真空开		
						arrCyCtrl[arrCyNo.ElectValveName.AnDTCarryingVacuum].Cmd.bOFF:=TRUE;//叠台搬运真空开	
						arrCyCtrl[arrCyNo.ElectValveName.AndeviationVacuum].Cmd.bON:=FALSE;//纠偏平台真空关
						arrCyCtrl[arrCyNo.ElectValveName.AndeviationVacuum].Cmd.bOFF:=TRUE;//纠偏平台真空关		
						arrCyCtrl[arrCyNo.ElectValveName.AndeviationVacuumBark].Cmd.bON:=TRUE;//纠偏平台破真空
						arrCyCtrl[arrCyNo.ElectValveName.AndeviationVacuumBark].Cmd.bOFF:=FALSE;//纠偏平台破开真空	
						//IF Mach_Control.An_b.An_deviationFalg THEN
							Mach_Control.An_b.An_DPCarryingFalg:=TRUE;//复位负极送片搬运吸盘上有料标记
							Mach_Control.An_b.An_deviationFalg:=FALSE;//置位纠偏平台上有料标记
						//END_IF
						Par.stDT_date.An_MQ_Slice[2]:=Par.stDT_date.An_MQ_Slice[1];
				
				 An_StandbyStep2:=666;
			END_IF	
			


400:    
				IF arrAxisCtrl[AxiseNo.VirAxisName.VirMain].Status.fActPos>=250  AND arrAxisCtrl[AxiseNo.VirAxisName.VirMain].Status.fActPos<=(250+6) AND NOT Mach_Control.An_b.An_MainBelting THEN   
								 IF (Mach_Control.An_b.An_MainBeltOK  OR  Mach_Control.U.EmptyRunMode ) AND NOT Mach_Control.An_b.An_CarryingFalg (*AND NOT Mach_Control.An_b.JumpPiceReady*)  THEN
									arrCyCtrl[arrCyNo.ElectValveName.AnCarryingVacuum].Cmd.bON:=TRUE;////搬运真空			
									arrCyCtrl[arrCyNo.ElectValveName.AnCarryingVacuum].Cmd.bOFF:=FALSE;////搬运真空						
								   //  Mach_Control.An_b.An_MainBelting:=TRUE;//正极搬运升降取极片中	 
									 An_Step0:=10;  //调用升降取片流程 
							     ELSE
									 	//fbAnCamInCarryingUpDown.bCamInExecute:=FALSE;//正极升解除耦合
										Mach_Control.An_b.An_MainBelting:=FALSE;//正极搬运升降取极片中	
										arrCyCtrl[arrCyNo.ElectValveName.AnCarryingVacuum].Cmd.bON:=FALSE;////搬运真空			
										arrCyCtrl[arrCyNo.ElectValveName.AnCarryingVacuum].Cmd.bOFF:=FALSE;////搬运真空			
										arrCyCtrl[arrCyNo.ElectValveName.AnCarryingVacuumBark].Cmd.bON:=FALSE;////搬运破真空			
										arrCyCtrl[arrCyNo.ElectValveName.AnCarryingVacuumBark].Cmd.bOFF:=FALSE;////搬运破真空																		
										IF NOT arrAxisCtrl[AxiseNo.AxisName.AnCarryingUpDown].Cmd.arrbRealPoint[4] THEN
											arrAxisCtrl[AxiseNo.AxisName.AnCarryingUpDown].Cmd.iGoSetPos:=4;//移动至流水线上方
										END_IF	
							    END_IF	
		
				            An_StandbyStep2:=666;
				END_IF


(************************************NG纠偏流程*********************************************)
600:		//负极搬运放片到纠偏平台
			IF 	arrAxisCtrl[AxiseNo.VirAxisName.VirMain].Status.fActPos>=260  AND  arrAxisCtrl[AxiseNo.VirAxisName.VirMain].Status.fActPos<=320  THEN//198	
						arrCyCtrl[arrCyNo.ElectValveName.AnDTCarryingVacuumBark].Cmd.bON:=TRUE;	//正极叠台搬运升降真空	真空
						arrCyCtrl[arrCyNo.ElectValveName.AnDTCarryingVacuumBark].Cmd.bOFF:=FALSE;	//正极叠台搬运升降真空破真空											
						arrCyCtrl[arrCyNo.ElectValveName.AndeviationVacuum].Cmd.bON:=TRUE;	//正极纠偏台真空			
						arrCyCtrl[arrCyNo.ElectValveName.AndeviationVacuum].Cmd.bOFF:=FALSE;	//正极纠偏台真空
					//IF Mach_Control.An_b.An_CarryingFalg THEN	               
						Mach_Control.An_b.An_deviationFalg:=TRUE;//置位纠偏平台上有料标记 
						Mach_Control.An_b.An_CarryingFalg:=FALSE;//复位负极送片搬运吸盘上有料标记				
					//END_IF
					Par.stDT_date.An_MQ_Slice[1]:=Par.stDT_date.An_MQ_Slice[0];
			          An_StandbyStep2:=666;
		    END_IF					
				
END_CASE			

CASE An_StandbyStep3 OF 
	
100://		
	IF arrAxis[AxiseNo.VirAxisName.VirMain].NcToPlc.SetPos=360 AND  arrAxis[AxiseNo.VirAxisName.VirMain].Status.NotMoving  THEN
		arrCyCtrl[arrCyNo.ElectValveName.AndeviationIonizedWind].Cmd.bON:=TRUE;//正极纠偏平台除尘
		arrCyCtrl[arrCyNo.ElectValveName.AndeviationIonizedWind].Cmd.bOFF:=FALSE;//正极纠偏平台除尘
		DT_SingeMode();//单步选择		
		DP_Step1:=100;//解耦
		An_StandbyStep3:=110;
	END_IF;			
 110:
	IF DP_Step1=6666 THEN
		An_StandbyStep1:=1000;	
		An_StandbyStep3:=6666;
	END_IF	


	200:	
	IF arrAxis[AxiseNo.VirAxisName.VirMain].NcToPlc.SetPos=360 AND  arrAxis[AxiseNo.VirAxisName.VirMain].Status.NotMoving  THEN
		//	Mach_Control.Ca_b.Ca_CacheBelting:=FALSE;//负极搬运升降取极片中	
		DT_SingeMode();//单步选择
		DP_Step1:=100;
		An_StandbyStep3:=210;
	END_IF;								
     210:
               IF DP_Step1=6666 THEN
                  	An_StandbyStep1:=1000;		
			An_StandbyStep3:=6666;
               END_IF

300:
	IF arrAxis[AxiseNo.VirAxisName.VirMain].NcToPlc.SetPos=360 AND  arrAxis[AxiseNo.VirAxisName.VirMain].Status.NotMoving  THEN
		DT_SingeMode();//单步选择			
		DP_Step1:=100;
		An_StandbyStep3:=320;
	END_IF	
320:		
          IF DP_Step1=6666 	 THEN	
			     An_StandbyStep1:=1000;	
			      An_StandbyStep3:=6666;
	     END_IF;			


400:
      	IF arrAxis[AxiseNo.VirAxisName.VirMain].NcToPlc.SetPos=360 AND  arrAxis[AxiseNo.VirAxisName.VirMain].Status.NotMoving  THEN
					   DT_SingeMode();//单步选择			
                     	DP_Step1:=100;
						An_StandbyStep3:=420;
		END_IF		
								
420:		
                IF DP_Step1=6666 THEN	
						An_StandbyStep1:=1000;	
						An_StandbyStep3:=6666;
				END_IF;		

				
600:
      	IF arrAxis[AxiseNo.VirAxisName.VirMain].NcToPlc.SetPos=360 AND  arrAxis[AxiseNo.VirAxisName.VirMain].Status.NotMoving  THEN
				DT_SingeMode();//单步选择			
                DP_Step1:=100;
				An_StandbyStep3:=620; 
		END_IF		
								
620:		
                  IF DP_Step1=6666 THEN	
						//Ca_StandbyStep0:=1000;	
						An_StandbyStep3:=6666;
				END_IF;			
				
END_CASE
END_ACTION

ACTION An_StandbySub1:
An_TON[9].IN:=Mach_Control.An_b.bAn_PoleHave;
IF An_TON[9].Q THEN
	Mach_Control.An_b.bAn_PoleHave:=FALSE;//正极取流水线极片完成，
END_IF

//取料中信号复位
An_TON[10].IN:= NOT  arrAxisCtrl[AxiseNo.AxisName.AnCarryingUpDown].Cmd.arrbRealPoint[4] AND Mach_Control.An_b.JumpPiceReady AND Mach_Control.An_b.An_MainBelting;
IF An_TON[10].Q THEN
	IF NOT  arrAxisCtrl[AxiseNo.AxisName.AnCarryingUpDown].Cmd.arrbRealPoint[4] THEN		
		arrAxisCtrl[AxiseNo.AxisName.AnCarryingUpDown].Cmd.iGoSetPos:=4;//正极送片搬运升降上升至初始高度	
	ELSE
		arrAxisCtrl[AxiseNo.AxisName.AnCarryingUpDown].Cmd.iGoSetPos:=0;//正极送片搬运升降上升至初始高度	
	END_IF
END_IF
An_TON[11].IN:=arrAxisCtrl[AxiseNo.AxisName.AnCarryingUpDown].Cmd.arrbRealPoint[4] AND Mach_Control.An_b.JumpPiceReady AND Mach_Control.An_b.An_MainBelting;
IF An_TON[11].Q  THEN
	An_Step0:=0;
	Mach_Control.An_b.AN_BeltDone:=TRUE;//取流水线取极片完成
	Mach_Control.An_b.An_MainBelting:=FALSE;//正极搬运升降取极片中
END_IF



IF Mach_Control.U.DT_iMode=1 THEN//在自动状态下	
CASE An_Step0 OF

	10:
		IF arrAxisCtrl[AxiseNo.AxisName.AnCarryingLine].Status.Enabled AND arrAxisCtrl[AxiseNo.AxisName.AnCarryingUpDown].Status.Enabled
			AND arrAxisCtrl[AxiseNo.AxisName.AnCarryingWhirling].Status.Enabled THEN
		
			IF An_JumpRules[1] THEN//空叠隔膜 //OR An_JumpRules[3]  OR An_JumpRules[6] OR An_JumpRules[8] OR An_JumpRules[10]  
				An_Step0:=400;
			ELSE
				An_Step0:=50;
			END_IF
		END_IF
	50:

		//正极搬运升降上升至等待位  20240505 CF
		IF ABS(arrAxisCtrl[AxiseNo.AxisName.AnCarryingLine].Status.fSetPos-arrAxisPar[AxiseNo.AxisName.AnCarryingLine].arrTargetPoint[1])<0.5
			//AND arrAxisCtrl[AxiseNo.AxisName.AnCarryingUpDown].Cmd.arrbRealPoint[4] 					
			AND arrAxisCtrl[AxiseNo.AxisName.AnCarryingWhirling].Cmd.arrbRealPoint[1]  THEN
			IF Mach_Control.DT_b.SinStepMode THEN//单步调试模式
				DP_SinStepe:=TRUE;
			ELSE
				DP_SinStepe:=FALSE;	
			END_IF	
		An_Step0:=100;
		END_IF
	
	END_CASE
END_IF
arrAxisCtrl[AxiseNo.VirAxisName.VirMain].Status.fActPos;
CASE An_Step0 OF
	100://判断正极流水线是否允许取料
		IF NOT DP_SinStepe THEN
			IF (Mach_Control.An_b.An_MainBeltOK AND NOT Mach_Control.An_b.An_CarryingFalg)  OR  Mach_Control.U.EmptyRunMode THEN
				Mach_Control.An_b.An_MainBelting:=TRUE;//正极搬运升降取极片中
				IF Mach_Control.DT_b.SinStepMode THEN//单步调试模式
					DP_SinStepe:=TRUE;
				ELSE
					DP_SinStepe:=FALSE;	
				END_IF	
				An_TON[5].IN:=FALSE;			
				An_Step0:=150;
			ELSIF Mach_Control.An_b.An_CarryingFalg  THEN
				An_Step0:=6666;
			ELSIF NOT Mach_Control.U.EmptyRunMode AND  An_JumpRules[8] THEN
				An_Step0:=500;	
			ELSIF Mach_Control.An_b.JumpPiceReady AND NOT Mach_Control.An_b.An_MainBeltOK AND  DP_Step4=110 THEN
	            An_Step0:=0;
			END_IF
		END_IF
	150:
			IF NOT 	DP_SinStepe THEN				
				arrCyCtrl[arrCyNo.ElectValveName.AnCarryingVacuum].Cmd.bON:=TRUE;//正极搬运升降取料真空打开
				arrCyCtrl[arrCyNo.ElectValveName.AnCarryingVacuum].Cmd.bOFF:=FALSE;//正极搬运升降取料真空打开
				IF arrAxisCtrl[AxiseNo.AxisName.AnCarryingUpDown].Status.Homed(* AND arrAxisCtrl[AxiseNo.AxisName.AnCarryingUpDown].Status.NoMoving*) AND 
					NOT arrAxisCtrl[AxiseNo.AxisName.AnCarryingUpDown].Status.Error THEN
					IF arrAxisCtrl[AxiseNo.AxisName.AnCarryingUpDown].Cmd.arrbRealPoint[2] THEN	
							IF NOT An_TON[5].Q THEN
								An_TON[5].IN:=TRUE;
							ELSE
								arrAxisCtrl[AxiseNo.AxisName.AnCarryingUpDown].Cmd.iGoSetPos:=0;
								IF Mach_Control.DT_b.SinStepMode THEN//单步调试模式
									DP_SinStepe:=TRUE;
								ELSE
									DP_SinStepe:=FALSE;	
								END_IF		
								An_TON[5].IN:=FALSE;				
								An_Step0:=200;										
							END_IF									
					ELSE
						arrAxisCtrl[AxiseNo.AxisName.AnCarryingUpDown].Cmd.iGoSetPos:=2;//正极送片搬运升降下降至流水线取极片高度
					END_IF
				END_IF
			END_IF
	200:
	//20240414 wcz
	     IF   arrAxisCtrl[AxiseNo.AxisName.AnCarryingUpDown].Status.fActPos<=(arrAxisPar[AxiseNo.AxisName.AnCarryingUpDown].arrTargetPoint[2]-3)  AND 
			   arrAxisCtrl[AxiseNo.AxisName.AnCarryingUpDown].Status.Moving THEN
					Mach_Control.An_b.An_MainBelting:=FALSE;// 复位正极搬运升降取极片中
					Mach_Control.An_b.AN_BeltDone:=TRUE;//取流水线取极片完成
					Mach_Control.An_b.bAn_PoleHave:=TRUE;//正极取流水线极片完成，用来发给模切来清取料位极片有无信号
		 END_IF
	
		IF arrAxisCtrl[AxiseNo.AxisName.AnCarryingUpDown].Status.Homed (*AND arrAxisCtrl[AxiseNo.AxisName.AnCarryingUpDown].Status.NoMoving*) AND 
			NOT arrAxisCtrl[AxiseNo.AxisName.AnCarryingUpDown].Status.Error THEN
					IF arrAxisCtrl[AxiseNo.AxisName.AnCarryingUpDown].Cmd.arrbRealPoint[4] THEN
						arrAxisCtrl[AxiseNo.AxisName.AnCarryingUpDown].Cmd.iGoSetPos:=0;
						Mach_Control.An_b.An_MainBelting:=FALSE;// 复位正极搬运升降取极片中
						Mach_Control.An_b.AN_BeltDone:=TRUE;//取流水线取极片完成
						Mach_Control.An_b.An_CarryingFalg:=TRUE;//置位正极搬运升降真空吸盘上有极片
						Mach_Control.An_b.bAn_PoleHave:=TRUE;//正极取流水线极片完成，用来发给模切来清取料位极片有无信号
						Par.stDT_date.An_MQ_Slice[0]:=Par.stDT_date.AnMQ_MES;//转移皮带上的数据	
						An_Step0:=6666;
					ELSE
						arrAxisCtrl[AxiseNo.AxisName.AnCarryingUpDown].Cmd.iGoSetPos:=4;//正极送片搬运升降上升至初始高度
					END_IF
		END_IF	
	
		
	400:
		Mach_Control.An_b.An_MainBelting:=FALSE;// 复位正极搬运升降取极片中
		Mach_Control.An_b.AN_BeltDone:=TRUE;//取流水线取极片完成
		Mach_Control.An_b.An_CarryingFalg:=TRUE;//置位正极搬运升降真空吸盘上有极片
		//Par.stDT_date.An_MQ_Slice[0]:=Par.stDT_date.AnMQ_MES;//转移皮带上的数据	
		An_Step0:=6666;
		
	500:
		Mach_Control.An_b.An_MainBelting:=FALSE;// 复位正极搬运升降取极片中
		Mach_Control.An_b.AN_BeltDone:=TRUE;//取流水线取极片完成
		//Mach_Control.An_b.An_CarryingFalg:=TRUE;//置位正极搬运升降真空吸盘上有极片
		//Par.stDT_date.An_MQ_Slice[0]:=Par.stDT_date.AnMQ_MES;//转移皮带上的数据	
		An_Step0:=6666;
END_CASE

(*

//An_Step0--正极取流水线极片子程序
IF Mach_Control.U.DT_iMode=1 THEN//在自动状态下	
CASE An_Step0 OF
	10://正极搬运升降上升至等待位
		IF arrAxisCtrl[AxiseNo.AxisName.AnCarryingLine].Cmd.arrbRealPoint[1] 
		AND arrAxisCtrl[AxiseNo.AxisName.AnCarryingUpDown].Cmd.arrbRealPoint[4] 					
		AND arrAxisCtrl[AxiseNo.AxisName.AnCarryingWhirling].Cmd.arrbRealPoint[1]  THEN
			IF Mach_Control.DT_b.SinStepMode THEN//单步调试模式
				DP_SinStepe:=TRUE;
			ELSE
				DP_SinStepe:=FALSE;	
			END_IF	
		An_Step0:=30;
		END_IF
	30://判断正极流水线是否允许取料
		IF NOT DP_SinStepe THEN
				IF (Mach_Control.An_b.An_MainBeltOK AND NOT Mach_Control.An_b.An_CarryingFalg)  OR  Mach_Control.U.EmptyRunMode THEN
					Mach_Control.An_b.An_MainBelting:=TRUE;//正极搬运升降取极片中
					IF Mach_Control.DT_b.SinStepMode THEN//单步调试模式
						DP_SinStepe:=TRUE;
					ELSE
						DP_SinStepe:=FALSE;	
					END_IF	
					An_TON[5].IN:=FALSE;			
					An_Step0:=40;
				ELSIF Mach_Control.An_b.An_CarryingFalg  THEN
					An_Step0:=6666;
				(*
				ELSE
					An_Step0:=10;
					Mach_Control.An_b.An_MainBelting:=FALSE;//正极搬运升降取极片中
				*)
				END_IF
		END_IF
	(*
			IF NOT DP_SinStepe THEN
				IF  arrAxisCtrl[AxiseNo.AxisName.AnCarryingUpDown].Cmd.arrbRealPoint[4] AND arrAxisCtrl[AxiseNo.AxisName.AnCarryingUpDown].Status.Homed THEN
					An_Step0:=20;
				ELSE
						IF arrAxisCtrl[AxiseNo.AxisName.AnCarryingUpDown].Status.Homed AND arrAxisCtrl[AxiseNo.AxisName.AnCarryingUpDown].Status.NoMoving AND 
							NOT arrAxisCtrl[AxiseNo.AxisName.AnCarryingUpDown].Status.Error THEN
									IF arrAxisCtrl[AxiseNo.AxisName.AnCarryingUpDown].Cmd.arrbRealPoint[4] THEN
											arrAxisCtrl[AxiseNo.AxisName.AnCarryingUpDown].Cmd.iGoSetPos:=0;
											IF Mach_Control.DT_b.SinStepMode THEN//单步调试模式
												DP_SinStepe:=TRUE;
											ELSE
												DP_SinStepe:=FALSE;	
											END_IF						
											An_Step0:=20;
									ELSE
										arrAxisCtrl[AxiseNo.AxisName.AnCarryingUpDown].Cmd.iGoSetPos:=4;//正极送片搬运升降至等待高度
									END_IF
						END_IF
				END_IF
		END_IF;
	20://正极搬运平移至初始位，正极搬运旋转至初始位	
			IF NOT DP_SinStepe THEN	
					IF arrAxisCtrl[AxiseNo.AxisName.AnCarryingUpDown].Cmd.arrbRealPoint[4] AND arrAxisCtrl[AxiseNo.AxisName.AnCarryingLine].Status.Homed AND
						 arrAxisCtrl[AxiseNo.AxisName.AnCarryingLine].Status.NoMoving AND NOT arrAxisCtrl[AxiseNo.AxisName.AnCarryingLine].Status.Error THEN
								IF arrAxisCtrl[AxiseNo.AxisName.AnCarryingLine].Cmd.arrbRealPoint[1] THEN
									An_CarryingTorMark:=FALSE;//正极搬运1移位力矩判断标志位
									arrAxisCtrl[AxiseNo.AxisName.AnCarryingLine].Cmd.iGoSetPos:=0;
								ELSE
									arrAxisCtrl[AxiseNo.AxisName.AnCarryingLine].Cmd.iGoSetPos:=1;//正极搬运平移到初始位
									An_CarryingTorMark:=TRUE;//正极搬运1移位力矩判断标志位
								END_IF
					END_IF
					IF arrAxisCtrl[AxiseNo.AxisName.AnCarryingUpDown].Cmd.arrbRealPoint[4] AND arrAxisCtrl[AxiseNo.AxisName.AnCarryingWhirling].Status.Homed AND
						 arrAxisCtrl[AxiseNo.AxisName.AnCarryingWhirling].Status.NoMoving AND NOT arrAxisCtrl[AxiseNo.AxisName.AnCarryingWhirling].Status.Error THEN
								IF arrAxisCtrl[AxiseNo.AxisName.AnCarryingWhirling].Cmd.arrbRealPoint[1] THEN
									arrAxisCtrl[AxiseNo.AxisName.AnCarryingWhirling].Cmd.iGoSetPos:=0;
								ELSE
									arrAxisCtrl[AxiseNo.AxisName.AnCarryingWhirling].Cmd.iGoSetPos:=1;//正极搬运旋转至初始位
								END_IF
					END_IF
					IF arrAxisCtrl[AxiseNo.AxisName.AnCarryingLine].Cmd.arrbRealPoint[1] 
					AND arrAxisCtrl[AxiseNo.AxisName.AnCarryingUpDown].Cmd.arrbRealPoint[4] 					
					AND arrAxisCtrl[AxiseNo.AxisName.AnCarryingWhirling].Cmd.arrbRealPoint[1]  THEN
							IF Mach_Control.DT_b.SinStepMode THEN//单步调试模式
								DP_SinStepe:=TRUE;
							ELSE
								DP_SinStepe:=FALSE;	
							END_IF	
							An_Step0:=30;
					END_IF
			END_IF
	
		*)
	END_CASE
END_IF
arrAxisCtrl[AxiseNo.VirAxisName.VirMain].Status.fActPos;
CASE An_Step0 OF

	40:
			IF NOT 	DP_SinStepe THEN				
				arrCyCtrl[arrCyNo.ElectValveName.AnCarryingVacuum].Cmd.bON:=TRUE;//正极搬运升降取料真空打开
				arrCyCtrl[arrCyNo.ElectValveName.AnCarryingVacuum].Cmd.bOFF:=FALSE;//正极搬运升降取料真空打开
				IF arrAxisCtrl[AxiseNo.AxisName.AnCarryingUpDown].Status.Homed(* AND arrAxisCtrl[AxiseNo.AxisName.AnCarryingUpDown].Status.NoMoving*) AND 
					NOT arrAxisCtrl[AxiseNo.AxisName.AnCarryingUpDown].Status.Error THEN
					IF arrAxisCtrl[AxiseNo.AxisName.AnCarryingUpDown].Cmd.arrbRealPoint[2] THEN
							IF NOT An_TON[5].Q THEN
									An_TON[5].IN:=TRUE;
							ELSE
								arrAxisCtrl[AxiseNo.AxisName.AnCarryingUpDown].Cmd.iGoSetPos:=0;
								IF Mach_Control.DT_b.SinStepMode THEN//单步调试模式
									DP_SinStepe:=TRUE;
								ELSE
									DP_SinStepe:=FALSE;	
								END_IF		
								An_TON[5].IN:=FALSE;				
								An_Step0:=50;										
							END_IF									
					ELSE
						arrAxisCtrl[AxiseNo.AxisName.AnCarryingUpDown].Cmd.iGoSetPos:=2;//正极送片搬运升降下降至流水线取极片高度
					END_IF
				END_IF
			END_IF
50:
		IF arrAxisCtrl[AxiseNo.AxisName.AnCarryingUpDown].Status.Homed (*AND arrAxisCtrl[AxiseNo.AxisName.AnCarryingUpDown].Status.NoMoving*) AND 
			NOT arrAxisCtrl[AxiseNo.AxisName.AnCarryingUpDown].Status.Error THEN
					IF arrAxisCtrl[AxiseNo.AxisName.AnCarryingUpDown].Cmd.arrbRealPoint[4] THEN
						arrAxisCtrl[AxiseNo.AxisName.AnCarryingUpDown].Cmd.iGoSetPos:=0;
						Mach_Control.An_b.An_MainBelting:=FALSE;// 复位正极搬运升降取极片中
						Mach_Control.An_b.AN_BeltDone:=TRUE;//取流水线取极片完成
						Mach_Control.An_b.An_CarryingFalg:=TRUE;//置位正极搬运升降真空吸盘上有极片
						Par.stDT_date.An_MQ_Slice[0]:=Par.stDT_date.AnMQ_MES;//转移皮带上的数据	
						An_Step0:=6666;
					ELSE
						arrAxisCtrl[AxiseNo.AxisName.AnCarryingUpDown].Cmd.iGoSetPos:=4;//正极送片搬运升降上升至初始高度
					END_IF
		END_IF	

END_CASE

*)
END_ACTION

ACTION An_StandbySub2:
IF Mach_Control.U.DT_iMode=1 THEN//在自动状态下	
//An_Step1---正极送片搬运放片到纠偏台
	CASE An_Step1 OF

10:// 
	IF arrAxisCtrl[AxiseNo.AxisName.AnCarryingLine].Status.Enabled AND arrAxisCtrl[AxiseNo.AxisName.AnCarryingWhirling].Status.Enabled AND  arrAxisCtrl[AxiseNo.AxisName.AnCarryingUpDown].Status.Enabled  THEN
		IF arrAxisCtrl[AxiseNo.AxisName.AnCarryingLine].Cmd.arrbRealPoint[2]  AND  arrAxisCtrl[AxiseNo.AxisName.AnCarryingWhirling].Cmd.arrbRealPoint[2]   THEN
			An_Step1:=30;
		END_IF
	END_IF	
30://判断纠偏平台是否允许取极片
	IF NOT DP_SinStepe THEN
		DT_SingeMode();//单步选择			
		IF arrAxisCtrl[AxiseNo.AxisName.AnCarryingUpDown].Cmd.arrbRealPoint[3] THEN
			arrAxisCtrl[AxiseNo.AxisName.AnCarryingUpDown].Cmd.iGoSetPos:=0;
			/// 吸盘破真空    纠偏台开真空
			arrCyCtrl[arrCyNo.ElectValveName.AnCarryingVacuum].Cmd.bON:=FALSE;	//正极叠台搬运升降真空	真空
			arrCyCtrl[arrCyNo.ElectValveName.AnCarryingVacuum].Cmd.bOFF:=TRUE;	//正极叠台搬运升降真空破真空		
			arrCyCtrl[arrCyNo.ElectValveName.AnCarryingVacuumBark].Cmd.bON:=TRUE;	//正极叠台搬运升降真空	真空
			arrCyCtrl[arrCyNo.ElectValveName.AnCarryingVacuumBark].Cmd.bOFF:=FALSE;	//正极叠台搬运升降真空破真空											
			arrCyCtrl[arrCyNo.ElectValveName.AndeviationVacuum].Cmd.bON:=TRUE;	//正极纠偏台真空			
			arrCyCtrl[arrCyNo.ElectValveName.AndeviationVacuum].Cmd.bOFF:=FALSE;	//正极纠偏台真空	           
			An_Step1:=40;
		ELSE
			arrAxisCtrl[AxiseNo.AxisName.AnCarryingUpDown].Cmd.iGoSetPos:=3;//负极搬运升降2上升至凸轮耦合初始高度
		END_IF	
	END_IF
					
40:		
	IF NOT DP_SinStepe THEN
		IF arrAxisCtrl[AxiseNo.AxisName.AnCarryingUpDown].Cmd.arrbRealPoint[4] THEN
			arrAxisCtrl[AxiseNo.AxisName.AnCarryingUpDown].Cmd.iGoSetPos:=0;
			/// 吸盘破真空    纠偏台开真空
			arrCyCtrl[arrCyNo.ElectValveName.AnDTCarryingVacuum].Cmd.bON:=FALSE;	//正极叠台搬运升降真空
			arrCyCtrl[arrCyNo.ElectValveName.AnDTCarryingVacuum].Cmd.bOFF:=FALSE;	//正极叠台搬运升降真空
			arrCyCtrl[arrCyNo.ElectValveName.AnDTCarryingVacuumBark].Cmd.bON:=FALSE;	//正极叠台搬运升降破真空	
			arrCyCtrl[arrCyNo.ElectValveName.AnDTCarryingVacuumBark].Cmd.bOFF:=FALSE;	//正极叠台搬运升降破真空	
			//IF Mach_Control.An_b.An_CarryingFalg THEN
			Mach_Control.An_b.An_deviationFalg:=TRUE;//复位纠偏平台有料标记
			Mach_Control.An_b.An_CarryingFalg:=FALSE;//负极搬运真空吸盘有料标记复位
			//END_IF
			Par.stDT_date.An_MQ_Slice[1]:=Par.stDT_date.An_MQ_Slice[0];
			An_Step1:=6666;
		ELSE
			arrAxisCtrl[AxiseNo.AxisName.AnCarryingUpDown].Cmd.iGoSetPos:=4;//负极搬运升降2上升至凸轮耦合初始高度
		END_IF			
	END_IF

	END_CASE
END_IF
END_ACTION

ACTION An_StandbySub3:
 An_StandbySub3_ton[1](PT:=T#300MS);
An_StandbySub3_ton[2](PT:=T#250MS);
An_StandbySub3_ton[3](PT:=T#300MS);
An_NG_TON(IN:= , PT:=T#0.3S , Q=> , ET=> );
An_NG_TON2(IN:= , PT:=T#0.3S , Q=> , ET=> );
YS(IN:= , PT:=T#2S , Q=> , ET=> );
YS1(IN:= , PT:=T#0.3S , Q=> , ET=> );

//An_Step2------正极纠偏平台踢NG片子程序

IF Mach_Control.U.DT_iMode=1 OR avg1 THEN//在自动状态下	
//正极纠偏平台踢NG片子程序
CASE An_Step2 OF
	10:
		IF arrAxisCtrl[AxiseNo.AxisName.AnDTCarryingUpDown].Status.Enabled AND  arrAxisCtrl[AxiseNo.AxisName.AnDTCarryingLine].Status.Enabled THEN
			IF   arrCyCtrl[arrCyNo.ElectValveName.AnDTCarryingVacuum].Io.DIOnSwitch  THEN
				An_Step2:=12;
			ELSE
				//Mach_Control.An_b.Error[4] :=TRUE;//正极叠台搬运升降有极片，无真空信号报警
				An_StandbySub3_ton[3].IN:=FALSE;
				An_Step2:=11; 
				arrCyCtrl[arrCyNo.ElectValveName.AnDTCarryingVacuum].Cmd.bOFF:=FALSE;//正极叠片搬运升降真空关
				arrCyCtrl[arrCyNo.ElectValveName.AnDTCarryingVacuum].Cmd.bON:=TRUE;//正极叠片搬运升降真空关
				arrCyCtrl[arrCyNo.ElectValveName.AnDTCarryingVacuumBark].Cmd.bON:=TRUE;//正极叠片搬运破真空开
				arrCyCtrl[arrCyNo.ElectValveName.AnDTCarryingVacuumBark].Cmd.bOFF:=FALSE;//正极叠片搬运破真空关			  
			END_IF
	 	END_IF
    11:	 
	    An_StandbySub3_ton[3].IN:=TRUE;
		IF  An_StandbySub3_ton[3].Q THEN
			   An_Step2:=12; 
			   An_StandbySub3_ton[3].IN:=FALSE;
		END_IF
				
	12://正极NG收料气缸伸出	
			arrCyCtrl[arrCyNo.CylinderName.AnScrapbinCy].Cmd.bON:=TRUE;//正极纠偏气缸伸出
			IF  arrCyCtrl[arrCyNo.CylinderName.AnScrapbinCy].Status.ONState THEN
				An_Step2:=20;
				//An_Step4:=1000;
			END_IF
	20://正极搬运升降上升至初始位,正极叠片搬运升降至初始位
				IF NOT DP_SinStepe THEN	
					IF arrAxisCtrl[AxiseNo.AxisName.AnDTCarryingUpDown].Status.Homed AND arrAxisCtrl[AxiseNo.AxisName.AnDTCarryingUpDown].Status.NoMoving AND 
						NOT arrAxisCtrl[AxiseNo.AxisName.AnDTCarryingUpDown].Status.Error THEN
						IF arrAxisCtrl[AxiseNo.AxisName.AnDTCarryingUpDown].Cmd.arrbRealPoint[5] THEN
							arrAxisCtrl[AxiseNo.AxisName.AnDTCarryingUpDown].Cmd.iGoSetPos:=0;
						ELSE
							arrAxisCtrl[AxiseNo.AxisName.AnDTCarryingUpDown].Cmd.iGoSetPos:=5;//正极叠片平台升降上升避让高度
						END_IF
					END_IF
					IF 	arrAxisCtrl[AxiseNo.AxisName.AnDTCarryingUpDown].Cmd.arrbRealPoint[5] AND arrAxisCtrl[AxiseNo.AxisName.AnDTCarryingUpDown].Status.Homed THEN
						IF Mach_Control.DT_b.SinStepMode THEN//单步调试模式
							DP_SinStepe:=TRUE;
						ELSE
							DP_SinStepe:=FALSE;	
						END_IF				
						An_Step2:=40;
					END_IF	
				END_IF
	30://正极搬运平移回初始位
			IF NOT DP_SinStepe THEN
					IF arrAxisCtrl[AxiseNo.AxisName.AnCarryingUpDown].Cmd.arrbRealPoint[4] AND arrAxisCtrl[AxiseNo.AxisName.AnCarryingLine].Status.Homed AND arrCyCtrl[arrCyNo.CylinderName.AnScrapbinCy].Status.ONState  AND
						 arrAxisCtrl[AxiseNo.AxisName.AnCarryingLine].Status.NoMoving AND NOT arrAxisCtrl[AxiseNo.AxisName.AnCarryingLine].Status.Error THEN
								IF arrAxisCtrl[AxiseNo.AxisName.AnCarryingLine].Cmd.arrbRealPoint[1] THEN
									arrAxisCtrl[AxiseNo.AxisName.AnCarryingLine].Cmd.iGoSetPos:=0;
									IF Mach_Control.DT_b.SinStepMode THEN//单步调试模式
										DP_SinStepe:=TRUE;
									ELSE
										DP_SinStepe:=FALSE;	
									END_IF							
									An_Step2:=40;
								ELSE
									arrAxisCtrl[AxiseNo.AxisName.AnCarryingLine].Cmd.iGoSetPos:=1;//正极搬运平移到初始位
								END_IF
					END_IF
			END_IF
	40://正极叠台搬运平移至取片位
			IF NOT DP_SinStepe THEN
					IF arrAxisCtrl[AxiseNo.AxisName.AnDTCarryingUpDown].Cmd.arrbRealPoint[5] AND arrAxisCtrl[AxiseNo.AxisName.AnDTCarryingLine].Status.Homed AND
						 arrAxisCtrl[AxiseNo.AxisName.AnDTCarryingLine].Status.NoMoving AND NOT arrAxisCtrl[AxiseNo.AxisName.AnDTCarryingLine].Status.Error THEN
								IF arrAxisCtrl[AxiseNo.AxisName.AnDTCarryingLine].Cmd.arrbRealPoint[1] THEN
									arrAxisCtrl[AxiseNo.AxisName.AnDTCarryingLine].Cmd.iGoSetPos:=0;
									IF Mach_Control.DT_b.SinStepMode THEN//单步调试模式
										DP_SinStepe:=TRUE;
									ELSE
										DP_SinStepe:=FALSE;	
									END_IF	
									An_Step2:=45;
								ELSE
									arrAxisCtrl[AxiseNo.AxisName.AnDTCarryingLine].Cmd.iGoSetPos:=1;//正极叠台搬运平移至取片位
								END_IF
					END_IF	
			END_IF
			
	45:
		//IF  CCD.AnRec.Finish.RectifyResult<>1 THEN
		
			An_Step2:=50;
		//END_IF
		(*
			IF Mach_Control.An_b.An_Rectifydev_CS>=1 OR CCD.AnRec.Finish.RectifyResult=3 OR CCD.AnRec.Finish.RectifyResult=4  OR NOT Mach_Control.An_b.An_Rectifydev_PB THEN
				An_Step2:=50;
			ELSE
				An_Step2:=150;
			END_IF
		*)



	

		
	50://正极纠偏位NG料盒气缸伸出，正极叠片搬运升降轴下降至踢NG料高度     arrCyCtrl[arrCyNo.CylinderName.AnScrapbinCy].Status.OFFState
			IF NOT DP_SinStepe THEN		
				      	IF arrAxisCtrl[AxiseNo.AxisName.AnDTCarryingUpDown].Cmd.arrbRealPoint[5] THEN
						    arrCyCtrl[arrCyNo.CylinderName.AnScrapbinCy].Cmd.bOFF:=TRUE;//正极NG收纳盒气缸收回
						END_IF
						
						IF arrCyCtrl[arrCyNo.CylinderName.AnScrapbinCy].Status.OFFState AND An_NG_TON2.Q  THEN
								IF NOT An_NG_TON.Q THEN
											An_NG_TON.IN:=TRUE;
											Mach_Control.An_b.An_DPCarryingFalg:=FALSE;// 复位正极叠片搬运真空吸盘标记有料
											arrCyCtrl[arrCyNo.ElectValveName.AnDTCarryingVacuum].Cmd.bOFF:=FALSE;//正极叠片搬运升降真空关闭
											arrCyCtrl[arrCyNo.ElectValveName.AnDTCarryingVacuum].Cmd.bON:=TRUE;//正极叠片搬运升降真空关闭
											//arrCyCtrl[arrCyNo.ElectValveName.AnDTCarryingVacuumBark].Cmd.bON:=TRUE;//正极叠片搬运升降破真空打开		
											//arrCyCtrl[arrCyNo.ElectValveName.AnDTCarryingVacuumBark].Cmd.bOFF:=FALSE;//正极叠片搬运升降破真空打开		
								ELSE					
											IF Mach_Control.DT_b.SinStepMode THEN//单步调试模式
												DP_SinStepe:=TRUE;
											ELSE
												DP_SinStepe:=FALSE;	
											END_IF	
											An_NG_TON.IN:=FALSE;
											An_Step2:=60;
											An_CCDNG:=An_CCDNG+1;
								END_IF
						ELSE
							An_NG_TON2.IN:=TRUE;
						END_IF
			END_IF	
	60://NG气缸伸出
				IF NOT DP_SinStepe THEN	
						An_NG_TON2.IN:=FALSE;
						IF arrAxisCtrl[AxiseNo.AxisName.AnDTCarryingUpDown].Cmd.arrbRealPoint[5] THEN
					    	arrCyCtrl[arrCyNo.CylinderName.AnScrapbinCy].Cmd.bON:=TRUE;//正极纠偏气缸伸出
						END_IF
						
						IF  arrCyCtrl[arrCyNo.CylinderName.AnScrapbinCy].Status.ONState THEN
							IF Mach_Control.DT_b.SinStepMode THEN//单步调试模式
								DP_SinStepe:=TRUE;
							ELSE
								DP_SinStepe:=FALSE;	
							END_IF	
							An_Step2:=70;
						END_IF	
				END_IF	
	70://正极叠片搬运升降至初始位
		IF arrAxisCtrl[AxiseNo.AxisName.AnDTCarryingUpDown].Status.Homed AND arrAxisCtrl[AxiseNo.AxisName.AnDTCarryingUpDown].Status.NoMoving AND 
			NOT arrAxisCtrl[AxiseNo.AxisName.AnDTCarryingUpDown].Status.Error THEN
					IF arrAxisCtrl[AxiseNo.AxisName.AnDTCarryingUpDown].Cmd.arrbRealPoint[4] THEN
						arrAxisCtrl[AxiseNo.AxisName.AnDTCarryingUpDown].Cmd.iGoSetPos:=0;
						An_Step2:=80;
					ELSE
						arrAxisCtrl[AxiseNo.AxisName.AnDTCarryingUpDown].Cmd.iGoSetPos:=4;//正极叠片平台升降至等待位
					END_IF
		END_IF

	80:
	   IF HMI_Hour>=8 AND HMI_Hour<20 THEN
		  Par.stDT_date.An_Rectifydev_DayNG:=Par.stDT_date.An_Rectifydev_DayNG+1; 
	   END_IF
	
	   IF (HMI_Hour>=0 AND HMI_Hour<8) OR  (HMI_Hour>=20 AND HMI_Hour<=23) THEN
		 Par.stDT_date.An_Rectifydev_NightNG:=Par.stDT_date.An_Rectifydev_NightNG+1;
	   END_IF
	
		Par.stDT_date.An_Rectifydev_JS:=Par.stDT_date.An_Rectifydev_JS+1;
		Mach_Control.An_b.An_CCD_amount:=Mach_Control.An_b.An_CCD_amount+1;
		An_StandbySub3_ton[2].IN:=FALSE;
		Mach_Control.An_b.An_Rectifydev_CS:=0;
		An_Step2:=90;

	90:
		IF NOT Mach_Control.U.CCD_ChosesHMI  AND NOT  Mach_Control.U.EmptyRunMode AND An_OverNGStep=0 THEN												
					CCD.AnRec.Finish.RectifyResult:=0;
					CCD.AnRec.Finish.RectifyX1:=0;
					CCD.AnRec.Finish.RectifyX2:=0;
					CCD.AnRec.Finish.RectifyY:=0;												
					Mach_Control.An_b.An_CCDStart :=TRUE;//启动CCD拍照
					CCD.AnRec.Start.iPhotoDo:=1;//第二次拍照
					Mach_Control.An_b.An_VacuumErrorNG:=FALSE;
					An_Step2:=100;
		ELSE
					An_Step2:=6666;
		END_IF	
	100:
		IF NOT An_StandbySub3_ton[2].Q THEN
			An_StandbySub3_ton[2].IN:=TRUE;
		ELSE
			IF CCD.AnRec.Finish.RectifyResult<> 3 AND NOT Mach_Control.U.CCD_ChosesHMI THEN
				Mach_Control.An_b.Error[24]:=TRUE;//正极纠偏平台NG片未排掉报警，请拿掉
				An_StandbySub3_ton[2].IN:=FALSE;
				An_Step2:=6666;
			ELSE
				An_StandbySub3_ton[2].IN:=FALSE;
				An_Step2:=6666;
			END_IF
		END_IF
	



	
	//////////////////////////////////二次纠偏流程/////////////////////////////////////////////
	150:
		IF arrAxisCtrl[AxiseNo.AxisName.AndeviationX1].Cmd.arrbRealPoint[1] AND arrAxisCtrl[AxiseNo.AxisName.AndeviationX2].Cmd.arrbRealPoint[1]  
			AND arrAxisCtrl[AxiseNo.AxisName.AndeviationY].Cmd.arrbRealPoint[1]  THEN
			An_Step2:=160;
		END_IF
	
